//     normal_speed_task Inputs/csp_transfer_main_drives.SD41700_drv.channel_a.process_data_input.status_parametrization_level <-> AT 1/Status parametrization level
//     normal_speed_task Inputs/csp_transfer_main_drives.SD41700_drv.channel_a.process_data_input.warning_active <-> AT 1/Device control: Status word[2]
//     normal_speed_task Inputs/csp_transfer_main_drives.SD41700_drv.channel_b.process_data_input.status_parametrization_level <-> AT 1/Status parametrization level
//   SFI_CasePacker Instance <-> Transfer EtherCAT Master/Slot 57 (EK1100)/SPLC40210
//     highest_speed_task Inputs/csp_transfer_main_safety_drives_SD41100.chA_smes_sis.safely_closed_input.status <-> StandardInputs/SD41100.csp_transfer_main_safety_drives_SD41100chA_smes_sissafely_closed_inputstatus_31
//     highest_speed_task Inputs/csp_transfer_main_safety_drives_SD41300.chA_smes_sis.safely_closed_input.status <-> StandardInputs/SD41300.csp_transfer_main_safety_drives_SD41300chA_smes_sissafely_closed_inputstatus_61
//     highest_speed_task Inputs/csp_transfer_main_safety_drives_SD41400.chA_smes_sis.safely_closed_input.status <-> StandardInputs/SD41400.csp_transfer_main_safety_drives_SD41400chA_smes_sissafely_closed_inputstatus_69
//     highest_speed_task Inputs/csp_transfer_main_safety_drives_SD41500.chA_smes_sis.safely_closed_input.status <-> StandardInputs/SD41500.csp_transfer_main_safety_drives_SD41500chA_smes_sissafely_closed_inputstatus_77
//     highest_speed_task Inputs/csp_transfer_main_safety_drives_SD41100.chB_smes_sis.safely_closed_input.status <-> StandardInputs/SD41100.csp_transfer_main_safety_drives_SD41100chB_smes_sissafely_closed_inputstatus_32
//     highest_speed_task Inputs/csp_transfer_main_safety_drives_SD41300.chB_smes_sis.safely_closed_input.status <-> StandardInputs/SD41300.csp_transfer_main_safety_drives_SD41300chB_smes_sissafely_closed_inputstatus_62
//     highest_speed_task Inputs/csp_transfer_main_safety_drives_SD41400.chB_smes_sis.safely_closed_input.status <-> StandardInputs/SD41400.csp_transfer_main_safety_drives_SD41400chB_smes_sissafely_closed_inputstatus_70
//     highest_speed_task Inputs/csp_transfer_main_safety_drives_SD41500.chB_smes_sis.safely_closed_input.status <-> StandardInputs/SD41500.csp_transfer_main_safety_drives_SD41500chB_smes_sissafely_closed_inputstatus_78
//     highest_speed_task Inputs/csp_transfer_main_safety_guards.sis.safely_closed_input.status <-> StandardInputs/Guards.csp_transfer_main_safety_guardssissafely_closed_inputstatus_124
//     low_speed_task Inputs/csp_transfer_main_safety_accUChange.sig.group_info_data.info_data <-> TwinSAFE Group Info Data/AccUChange_STO Info Data
//     low_speed_task Inputs/csp_transfer_main_safety_accUChange.sis.discrepancy_input.status <-> StandardInputs/AccUChange_STO.csp_transfer_main_safety_accUChangesisdiscrepancy_inputstatus_169
//     low_speed_task Inputs/csp_transfer_main_safety_accUChange.sis.safely_closed_input.status <-> StandardInputs/AccUChange_STO.csp_transfer_main_safety_accUChangesissafely_closed_inputstatus_162
//     low_speed_task Inputs/csp_transfer_main_safety_drives_PS41020.sig.group_info_data.info_data <-> TwinSAFE Group Info Data/DrivesRackPowerSupply Info Data
//     low_speed_task Inputs/csp_transfer_main_safety_drives_PS41020.sig.safety_group_fb_err_input.status <-> StandardInputs/DrivesRackPowerSupply.csp_transfer_main_safety_drives_PS41020sigsafety_group_fb_err_inputstatus_172
//     low_speed_task Inputs/csp_transfer_main_safety_drives_SD41200.chA_smes_sis.safely_closed_input.status <-> StandardInputs/SD41200.csp_transfer_main_safety_drives_SD41200chA_smes_sissafely_closed_inputstatus_50
//     low_speed_task Inputs/csp_transfer_main_safety_drives_SD41600.chA_smes_sis.safely_closed_input.status <-> StandardInputs/SD41600.csp_transfer_main_safety_drives_SD41600chA_smes_sissafely_closed_inputstatus_85
//     low_speed_task Inputs/csp_transfer_main_safety_drives_SD41700.chA_smes_sis.safely_closed_input.status <-> StandardInputs/SD41700.csp_transfer_main_safety_drives_SD41700chA_smes_sissafely_closed_inputstatus_93
//     low_speed_task Inputs/csp_transfer_main_safety_drives_SD41200.chB_smes_sis.safely_closed_input.status <-> StandardInputs/SD41200.csp_transfer_main_safety_drives_SD41200chB_smes_sissafely_closed_inputstatus_52
//     low_speed_task Inputs/csp_transfer_main_safety_drives_SD41600.chB_smes_sis.safely_closed_input.status <-> StandardInputs/SD41600.csp_transfer_main_safety_drives_SD41600chB_smes_sissafely_closed_inputstatus_86
//     low_speed_task Inputs/csp_transfer_main_safety_drives_SD41700.chB_smes_sis.safely_closed_input.status <-> StandardInputs/SD41700.csp_transfer_main_safety_drives_SD41700chB_smes_sissafely_closed_inputstatus_94
//     low_speed_task Inputs/csp_transfer_main_safety_drives_commonConfiguration.rack_smes_sis.safely_closed_input.status <-> StandardInputs/DrivesCommonConfiguration.csp_transfer_main_safety_drives_commonConfigurationrack_smes_sissafely_closed_inputstatus_28
//     low_speed_task Inputs/csp_transfer_main_safety_drives_commonConfiguration.sig.group_info_data.info_data <-> TwinSAFE Group Info Data/DrivesCommonConfiguration Info Data
//     low_speed_task Inputs/csp_transfer_main_safety_emergency.HMI_button_sio.protection_safely_closed_input.status <-> StandardInputs/Interface.csp_transfer_main_safety_emergencyHMI_button_stop_sioprotection_safely_closed_inputstatus_6
//     low_speed_task Inputs/csp_transfer_main_safety_emergency.delayed_sis.safely_closed_input.status <-> StandardInputs/EmergencyCircuit.csp_transfer_main_safety_emergencydelayed_sissafely_closed_inputstatus_111
//     low_speed_task Inputs/csp_transfer_main_safety_emergency.sig.group_info_data.info_data <-> TwinSAFE Group Info Data/EmergencyCircuit Info Data
//     low_speed_task Inputs/csp_transfer_main_safety_guards.delayed_sis.safely_closed_input.status <-> StandardInputs/Guards.csp_transfer_main_safety_guardsdelayed_sissafely_closed_inputstatus_114
//     low_speed_task Inputs/csp_transfer_main_safety_guards.sig.group_info_data.info_data <-> TwinSAFE Group Info Data/Guards Info Data
//     low_speed_task Inputs/csp_transfer_main_safety_guards.sio_door_3.protection_discrepancy_input.status <-> StandardInputs/Guards.csp_transfer_main_safety_guardssio_door_3protection_discrepancy_inputstatus_115
//     low_speed_task Inputs/csp_transfer_main_safety_guards.sio_door_4.protection_discrepancy_input.status <-> StandardInputs/Guards.csp_transfer_main_safety_guardssio_door_4protection_discrepancy_inputstatus_126
//     low_speed_task Inputs/csp_transfer_main_safety_guards.sio_door_5.protection_discrepancy_input.status <-> StandardInputs/Guards.csp_transfer_main_safety_guardssio_door_5protection_discrepancy_inputstatus_128
//     low_speed_task Inputs/csp_transfer_main_safety_guards.sio_door_6.protection_discrepancy_input.status <-> StandardInputs/Guards.csp_transfer_main_safety_guardssio_door_6protection_discrepancy_inputstatus_132
//     low_speed_task Inputs/csp_transfer_main_safety_guards.sio_door_7.protection_discrepancy_input.status <-> StandardInputs/Guards.csp_transfer_main_safety_guardssio_door_7protection_discrepancy_inputstatus_148
//     low_speed_task Inputs/csp_transfer_main_safety_guards.sio_door_8.protection_discrepancy_input.status <-> StandardInputs/Guards.csp_transfer_main_safety_guardssio_door_8protection_discrepancy_inputstatus_151
//     low_speed_task Inputs/csp_transfer_main_safety_guards.sio_door_3.safely_closed_and_locked_input.status <-> StandardInputs/Guards.csp_transfer_main_safety_guardssio_door_3safely_closed_and_locked_inputstatus_118
//     low_speed_task Inputs/csp_transfer_main_safety_guards.sio_door_4.safely_closed_and_locked_input.status <-> StandardInputs/Guards.csp_transfer_main_safety_guardssio_door_4safely_closed_and_locked_inputstatus_125
//     low_speed_task Inputs/csp_transfer_main_safety_guards.sio_door_5.safely_closed_and_locked_input.status <-> StandardInputs/Guards.csp_transfer_main_safety_guardssio_door_5safely_closed_and_locked_inputstatus_129
//     low_speed_task Inputs/csp_transfer_main_safety_guards.sio_door_6.safely_closed_and_locked_input.status <-> StandardInputs/Guards.csp_transfer_main_safety_guardssio_door_6safely_closed_and_locked_inputstatus_133
//     low_speed_task Inputs/csp_transfer_main_safety_guards.sio_door_7.safely_closed_and_locked_input.status <-> StandardInputs/Guards.csp_transfer_main_safety_guardssio_door_7safely_closed_and_locked_inputstatus_149
//     low_speed_task Inputs/csp_transfer_main_safety_guards.sio_door_8.safely_closed_and_locked_input.status <-> StandardInputs/Guards.csp_transfer_main_safety_guardssio_door_8safely_closed_and_locked_inputstatus_150
//     low_speed_task Inputs/csp_transfer_main_safety_guards.sio_door_3.safely_locked_input.status <-> StandardInputs/Guards.csp_transfer_main_safety_guardssio_door_3safely_locked_inputstatus_116
//     low_speed_task Inputs/csp_transfer_main_safety_guards.sio_door_4.safely_locked_input.status <-> StandardInputs/Guards.csp_transfer_main_safety_guardssio_door_4safely_locked_inputstatus_141
//     low_speed_task Inputs/csp_transfer_main_safety_guards.sio_door_5.safely_locked_input.status <-> StandardInputs/Guards.csp_transfer_main_safety_guardssio_door_5safely_locked_inputstatus_130
//     low_speed_task Inputs/csp_transfer_main_safety_guards.sio_door_6.safely_locked_input.status <-> StandardInputs/Guards.csp_transfer_main_safety_guardssio_door_6safely_locked_inputstatus_142
//     low_speed_task Inputs/csp_transfer_main_safety_guards.sio_door_7.safely_locked_input.status <-> StandardInputs/Guards.csp_transfer_main_safety_guardssio_door_7safely_locked_inputstatus_152
//     low_speed_task Inputs/csp_transfer_main_safety_guards.sio_door_8.safely_locked_input.status <-> StandardInputs/Guards.csp_transfer_main_safety_guardssio_door_8safely_locked_inputstatus_153
//     low_speed_task Inputs/csp_transfer_main_safety_token.sig.group_info_data.info_data <-> TwinSAFE Group Info Data/SafetyToken Info Data
//     low_speed_task Inputs/csp_transfer_main_safety_token.sio.protection_discrepancy_input.status <-> StandardInputs/SafetyToken.csp_transfer_main_safety_tokensioprotection_discrepancy_inputstatus_140
//     low_speed_task Inputs/csp_transfer_main_safety_token.sio.protection_safely_closed_input.status <-> StandardInputs/Interface.csp_transfer_main_safety_tokensioprotection_safely_closed_inputstatus_171
//     low_speed_task Inputs/csp_transfer_main_safety_token.sis.safely_closed_input.status <-> StandardInputs/SafetyToken.csp_transfer_main_safety_tokensissafely_closed_inputstatus_137
//     low_speed_task Outputs/csp_transfer_main_safety_accUChange.sig.safety_group_err_ack_output.status <-> StandardOutputs/AccUChange_STO.ErrorAcknowledgement_159
//     low_speed_task Outputs/csp_transfer_main_safety_accUChange.sig.safety_group_run_output.status <-> StandardOutputs/AccUChange_STO.Run_160
//     low_speed_task Outputs/csp_transfer_main_safety_accUChange.sis.open_output.status <-> StandardOutputs/AccUChange_STO.csp_transfer_main_safety_accUChangesisopen_outputstatus_161
//     low_speed_task Outputs/csp_transfer_main_safety_drives_PS41020.sig.safety_group_err_ack_output.status <-> StandardOutputs/DrivesRackPowerSupply.csp_transfer_main_safety_drives_PS41020sigsafety_group_err_ack_outputstatus_13
//     low_speed_task Outputs/csp_transfer_main_safety_drives_PS41020.sig.safety_group_run_output.status <-> StandardOutputs/DrivesRackPowerSupply.csp_transfer_main_safety_drives_PS41020sigsafety_group_run_outputstatus_14
//     low_speed_task Outputs/csp_transfer_main_safety_drives_SD41100.chA_smes_sis.open_output.status <-> StandardOutputs/SD41100.csp_transfer_main_safety_drives_SD41100chA_smes_sisopen_outputstatus_22
//     low_speed_task Outputs/csp_transfer_main_safety_drives_SD41200.chA_smes_sis.open_output.status <-> StandardOutputs/SD41200.csp_transfer_main_safety_drives_SD41200chA_smes_sisopen_outputstatus_49
//     low_speed_task Outputs/csp_transfer_main_safety_drives_SD41300.chA_smes_sis.open_output.status <-> StandardOutputs/SD41300.csp_transfer_main_safety_drives_SD41300chA_smes_sisopen_outputstatus_57
//     low_speed_task Outputs/csp_transfer_main_safety_drives_SD41400.chA_smes_sis.open_output.status <-> StandardOutputs/SD41400.csp_transfer_main_safety_drives_SD41400chA_smes_sisopen_outputstatus_65
//     low_speed_task Outputs/csp_transfer_main_safety_drives_SD41500.chA_smes_sis.open_output.status <-> StandardOutputs/SD41500.csp_transfer_main_safety_drives_SD41500chA_smes_sisopen_outputstatus_73
//     low_speed_task Outputs/csp_transfer_main_safety_drives_SD41600.chA_smes_sis.open_output.status <-> StandardOutputs/SD41600.csp_transfer_main_safety_drives_SD41600chA_smes_sisopen_outputstatus_81
//     low_speed_task Outputs/csp_transfer_main_safety_drives_SD41700.chA_smes_sis.open_output.status <-> StandardOutputs/SD41700.csp_transfer_main_safety_drives_SD41700chA_smes_sisopen_outputstatus_89
//     low_speed_task Outputs/csp_transfer_main_safety_drives_SD41100.chB_smes_sis.open_output.status <-> StandardOutputs/SD41100.csp_transfer_main_safety_drives_SD41100chB_smes_sisopen_outputstatus_23
//     low_speed_task Outputs/csp_transfer_main_safety_drives_SD41200.chB_smes_sis.open_output.status <-> StandardOutputs/SD41200.csp_transfer_main_safety_drives_SD41200chB_smes_sisopen_outputstatus_51
//     low_speed_task Outputs/csp_transfer_main_safety_drives_SD41300.chB_smes_sis.open_output.status <-> StandardOutputs/SD41300.csp_transfer_main_safety_drives_SD41300chB_smes_sisopen_outputstatus_58
//     low_speed_task Outputs/csp_transfer_main_safety_drives_SD41400.chB_smes_sis.open_output.status <-> StandardOutputs/SD41400.csp_transfer_main_safety_drives_SD41400chB_smes_sisopen_outputstatus_66
//     low_speed_task Outputs/csp_transfer_main_safety_drives_SD41500.chB_smes_sis.open_output.status <-> StandardOutputs/SD41500.csp_transfer_main_safety_drives_SD41500chB_smes_sisopen_outputstatus_74
//     low_speed_task Outputs/csp_transfer_main_safety_drives_SD41600.chB_smes_sis.open_output.status <-> StandardOutputs/SD41600.csp_transfer_main_safety_drives_SD41600chB_smes_sisopen_outputstatus_82
//     low_speed_task Outputs/csp_transfer_main_safety_drives_SD41700.chB_smes_sis.open_output.status <-> StandardOutputs/SD41700.csp_transfer_main_safety_drives_SD41700chB_smes_sisopen_outputstatus_90
//     low_speed_task Outputs/csp_transfer_main_safety_drives_commonConfiguration.rack_smes_sis.open_output.status <-> StandardOutputs/DrivesCommonConfiguration.csp_transfer_main_safety_drives_commonConfigurationrack_smes_sisopen_outputstatus_27
//     low_speed_task Outputs/csp_transfer_main_safety_drives_commonConfiguration.sig.safety_group_err_ack_output.status <-> StandardOutputs/DrivesCommonConfiguration.ErrorAcknowledgement_25
//     low_speed_task Outputs/csp_transfer_main_safety_drives_commonConfiguration.sig.safety_group_run_output.status <-> StandardOutputs/DrivesCommonConfiguration.Run_26
//     low_speed_task Outputs/csp_transfer_main_safety_emergency.delayed_sis.open_output.status <-> StandardOutputs/EmergencyCircuit.csp_transfer_main_safety_emergencydelayed_sisopen_outputstatus_110
//     low_speed_task Outputs/csp_transfer_main_safety_emergency.sig.safety_group_err_ack_output.status <-> StandardOutputs/EmergencyCircuit.csp_transfer_main_safety_emergencysigsafety_group_err_ack_outputstatus_1
//     low_speed_task Outputs/csp_transfer_main_safety_emergency.sig.safety_group_run_output.status <-> StandardOutputs/EmergencyCircuit.csp_transfer_main_safety_emergencysigsafety_group_run_outputstatus_2
//     low_speed_task Outputs/csp_transfer_main_safety_guards.delayed_sis.open_output.status <-> StandardOutputs/Guards.csp_transfer_main_safety_guardsdelayed_sisopen_outputstatus_119
//     low_speed_task Outputs/csp_transfer_main_safety_guards.sig.safety_group_err_ack_output.status <-> StandardOutputs/Guards.ErrorAcknowledgement_112
//     low_speed_task Outputs/csp_transfer_main_safety_guards.sig.safety_group_run_output.status <-> StandardOutputs/Guards.Run_113
//     low_speed_task Outputs/csp_transfer_main_safety_guards.sio_door_3.unlock_output.status <-> StandardOutputs/Guards.csp_transfer_main_safety_guardssio_door_3unlock_outputstatus_127
//     low_speed_task Outputs/csp_transfer_main_safety_guards.sio_door_4.unlock_output.status <-> StandardOutputs/Guards.csp_transfer_main_safety_guardssio_door_4unlock_outputstatus_143
//     low_speed_task Outputs/csp_transfer_main_safety_guards.sio_door_5.unlock_output.status <-> StandardOutputs/Guards.csp_transfer_main_safety_guardssio_door_5unlock_outputstatus_131
//     low_speed_task Outputs/csp_transfer_main_safety_guards.sio_door_6.unlock_output.status <-> StandardOutputs/Guards.csp_transfer_main_safety_guardssio_door_6unlock_outputstatus_144
//     low_speed_task Outputs/csp_transfer_main_safety_guards.sio_door_7.unlock_output.status <-> StandardOutputs/Guards.csp_transfer_main_safety_guardssio_door_7unlock_outputstatus_154
//     low_speed_task Outputs/csp_transfer_main_safety_guards.sio_door_8.unlock_output.status <-> StandardOutputs/Guards.csp_transfer_main_safety_guardssio_door_8unlock_outputstatus_155
//     low_speed_task Outputs/csp_transfer_main_safety_token.sig.safety_group_err_ack_output.status <-> StandardOutputs/SafetyToken.ErrorAcknowledgement_134
//     low_speed_task Outputs/csp_transfer_main_safety_token.sig.safety_group_run_output.status <-> StandardOutputs/SafetyToken.Run_135
//     low_speed_task Outputs/csp_transfer_main_safety_token.sis.open_output.status <-> StandardOutputs/SafetyToken.csp_transfer_main_safety_tokensisopen_outputstatus_138
//     normal_speed_task Inputs/csp_transfer_main_safety_drives_PS41020.sis.discrepancy_input.status <-> StandardInputs/DrivesRackPowerSupply.csp_transfer_main_safety_drives_PS41020sisdiscrepancy_inputstatus_24
//     normal_speed_task Inputs/csp_transfer_main_safety_drives_PS41020.sis.safely_closed_input.status <-> StandardInputs/DrivesRackPowerSupply.csp_transfer_main_safety_drives_PS41020sissafely_closed_inputstatus_16
//     normal_speed_task Inputs/csp_transfer_main_safety_drives_SD{41100..41700 step 100}.sig.group_info_data.info_data <-> TwinSAFE Group Info Data/SD{41100..41700 step 100} Info Data  (7 links)
//     normal_speed_task Inputs/csp_transfer_main_safety_drives_SD41100.sig.safety_group_com_err_input.status <-> StandardInputs/SD41100.csp_transfer_main_safety_drives_SD41100sigsafety_group_com_err_inputstatus_36
//     normal_speed_task Inputs/csp_transfer_main_safety_drives_SD41200.sig.safety_group_com_err_input.status <-> StandardInputs/SD41200.csp_transfer_main_safety_drives_SD41200sigsafety_group_com_err_inputstatus_53
//     normal_speed_task Inputs/csp_transfer_main_safety_drives_SD41300.sig.safety_group_com_err_input.status <-> StandardInputs/SD41300.csp_transfer_main_safety_drives_SD41300sigsafety_group_com_err_inputstatus_63
//     normal_speed_task Inputs/csp_transfer_main_safety_drives_SD41400.sig.safety_group_com_err_input.status <-> StandardInputs/SD41400.csp_transfer_main_safety_drives_SD41400sigsafety_group_com_err_inputstatus_71
//     normal_speed_task Inputs/csp_transfer_main_safety_drives_SD41500.sig.safety_group_com_err_input.status <-> StandardInputs/SD41500.csp_transfer_main_safety_drives_SD41500sigsafety_group_com_err_inputstatus_79
//     normal_speed_task Inputs/csp_transfer_main_safety_drives_SD41600.sig.safety_group_com_err_input.status <-> StandardInputs/SD41600.csp_transfer_main_safety_drives_SD41600sigsafety_group_com_err_inputstatus_88
//     normal_speed_task Inputs/csp_transfer_main_safety_drives_SD41700.sig.safety_group_com_err_input.status <-> StandardInputs/SD41700.csp_transfer_main_safety_drives_SD41700sigsafety_group_com_err_inputstatus_95
//     normal_speed_task Inputs/csp_transfer_main_safety_drives_SD41100.sig.safety_group_fb_err_input.status <-> StandardInputs/SD41100.csp_transfer_main_safety_drives_SD41100sigsafety_group_fb_err_inputstatus_35
//     normal_speed_task Inputs/csp_transfer_main_safety_drives_SD41200.sig.safety_group_fb_err_input.status <-> StandardInputs/SD41200.csp_transfer_main_safety_drives_SD41200sigsafety_group_fb_err_inputstatus_54
//     normal_speed_task Inputs/csp_transfer_main_safety_drives_SD41300.sig.safety_group_fb_err_input.status <-> StandardInputs/SD41300.csp_transfer_main_safety_drives_SD41300sigsafety_group_fb_err_inputstatus_64
//     normal_speed_task Inputs/csp_transfer_main_safety_drives_SD41400.sig.safety_group_fb_err_input.status <-> StandardInputs/SD41400.csp_transfer_main_safety_drives_SD41400sigsafety_group_fb_err_inputstatus_72
//     normal_speed_task Inputs/csp_transfer_main_safety_drives_SD41500.sig.safety_group_fb_err_input.status <-> StandardInputs/SD41500.csp_transfer_main_safety_drives_SD41500sigsafety_group_fb_err_inputstatus_80
//     normal_speed_task Inputs/csp_transfer_main_safety_drives_SD41600.sig.safety_group_fb_err_input.status <-> StandardInputs/SD41600.csp_transfer_main_safety_drives_SD41600sigsafety_group_fb_err_inputstatus_87
//     normal_speed_task Inputs/csp_transfer_main_safety_drives_SD41700.sig.safety_group_fb_err_input.status <-> StandardInputs/SD41700.csp_transfer_main_safety_drives_SD41700sigsafety_group_fb_err_inputstatus_96
//     normal_speed_task Inputs/csp_transfer_main_safety_emergency.HMI_button_sio.protection_discrepancy_input.status <-> StandardInputs/EmergencyCircuit.csp_transfer_main_safety_emergencyHMI_button_sioprotection_discrepancy_inputstatus_12
//     normal_speed_task Inputs/csp_transfer_main_safety_emergency.sis.safely_closed_input.status <-> StandardInputs/EmergencyCircuit.csp_transfer_main_safety_emergencysissafely_closed_inputstatus_11
//     normal_speed_task Inputs/csp_transfer_main_safety_interface.SPLC40210_sig.group_info_data.info_data <-> TwinSAFE Group Info Data/Interface Info Data
//     normal_speed_task Inputs/csp_transfer_main_safety_interface._SD41100_drv_ChA.connection_info_data_interface.info_data <-> Connection Info Data/SD41100.SD41100_ChA_33 Info Data
//     normal_speed_task Inputs/csp_transfer_main_safety_interface._SD41200_drv_ChA.connection_info_data_interface.info_data <-> Connection Info Data/SD41200.SD41200_ChA_97 Info Data
//     normal_speed_task Inputs/csp_transfer_main_safety_interface._SD41300_drv_ChA.connection_info_data_interface.info_data <-> Connection Info Data/SD41300.SD41300_ChA_99 Info Data
//     normal_speed_task Inputs/csp_transfer_main_safety_interface._SD41400_drv_ChA.connection_info_data_interface.info_data <-> Connection Info Data/SD41400.SD41400_ChA_101 Info Data
//     normal_speed_task Inputs/csp_transfer_main_safety_interface._SD41500_drv_ChA.connection_info_data_interface.info_data <-> Connection Info Data/SD41500.SD41500_ChA_103 Info Data
//     normal_speed_task Inputs/csp_transfer_main_safety_interface._SD41600_drv_ChA.connection_info_data_interface.info_data <-> Connection Info Data/SD41600.SD41600_ChA_105 Info Data
//     normal_speed_task Inputs/csp_transfer_main_safety_interface._SD41700_drv_ChA.connection_info_data_interface.info_data <-> Connection Info Data/SD41700.SD41700_ChA_107 Info Data
//     normal_speed_task Inputs/csp_transfer_main_safety_interface._SD41100_drv_ChB.connection_info_data_interface.info_data <-> Connection Info Data/SD41100.SD41100_ChB_34 Info Data
//     normal_speed_task Inputs/csp_transfer_main_safety_interface._SD41200_drv_ChB.connection_info_data_interface.info_data <-> Connection Info Data/SD41200.SD41200_ChB_98 Info Data
//     normal_speed_task Inputs/csp_transfer_main_safety_interface._SD41300_drv_ChB.connection_info_data_interface.info_data <-> Connection Info Data/SD41300.SD41300_ChB_100 Info Data
//     normal_speed_task Inputs/csp_transfer_main_safety_interface._SD41400_drv_ChB.connection_info_data_interface.info_data <-> Connection Info Data/SD41400.SD41400_ChB_102 Info Data
//     normal_speed_task Inputs/csp_transfer_main_safety_interface._SD41500_drv_ChB.connection_info_data_interface.info_data <-> Connection Info Data/SD41500.SD41500_ChB_104 Info Data
//     normal_speed_task Inputs/csp_transfer_main_safety_interface._SD41600_drv_ChB.connection_info_data_interface.info_data <-> Connection Info Data/SD41600.SD41600_ChB_106 Info Data
//     normal_speed_task Inputs/csp_transfer_main_safety_interface._SD41700_drv_ChB.connection_info_data_interface.info_data <-> Connection Info Data/SD41700.SD41700_ChB_108 Info Data
//     normal_speed_task Inputs/csp_transfer_main_safety_interface._SPLC40210Slot59.connection_info_data_interface.info_data <-> Connection Info Data/Interface.SPLC40210Slot59_156 Info Data
//     normal_speed_task Inputs/csp_transfer_main_safety_interface._SPLC40210Slot60.connection_info_data_interface.info_data <-> Connection Info Data/Interface.SPLC40210Slot60_109 Info Data
//     normal_speed_task Inputs/csp_transfer_main_safety_interface._SPLC40210Slot61.connection_info_data_interface.info_data <-> Connection Info Data/Interface.SPLC40210Slot61_136 Info Data
//     normal_speed_task Inputs/csp_transfer_main_safety_interface._SPLC40210Slot68.connection_info_data_interface.info_data <-> Connection Info Data/Interface.SPLC40210Slot68_145 Info Data
//     normal_speed_task Inputs/csp_transfer_main_safety_interface._SPLC40210Slot70.connection_info_data_interface.info_data <-> Connection Info Data/Interface.SPLC40210Slot70_146 Info Data
//     normal_speed_task Inputs/csp_transfer_main_safety_interface._SPLC40210Slot72.connection_info_data_interface.info_data <-> Connection Info Data/Interface.SPLC40210Slot72_147 Info Data
//     normal_speed_task Outputs/csp_transfer_main_safety_drives_PS41020.sis.open_output.status <-> StandardOutputs/DrivesRackPowerSupply.csp_transfer_main_safety_drives_PS41020sisopen_outputstatus_15
//     normal_speed_task Outputs/csp_transfer_main_safety_drives_SD41100.sig.safety_group_err_ack_output.status <-> StandardOutputs/SD41100.ErrorAcknowledgement_18
//     normal_speed_task Outputs/csp_transfer_main_safety_drives_SD41200.sig.safety_group_err_ack_output.status <-> StandardOutputs/SD41200.ErrorAcknowledgement_37
//     normal_speed_task Outputs/csp_transfer_main_safety_drives_SD41300.sig.safety_group_err_ack_output.status <-> StandardOutputs/SD41300.ErrorAcknowledgement_39
//     normal_speed_task Outputs/csp_transfer_main_safety_drives_SD41400.sig.safety_group_err_ack_output.status <-> StandardOutputs/SD41400.ErrorAcknowledgement_41
//     normal_speed_task Outputs/csp_transfer_main_safety_drives_SD41500.sig.safety_group_err_ack_output.status <-> StandardOutputs/SD41500.ErrorAcknowledgement_43
//     normal_speed_task Outputs/csp_transfer_main_safety_drives_SD41600.sig.safety_group_err_ack_output.status <-> StandardOutputs/SD41600.ErrorAcknowledgement_45
//     normal_speed_task Outputs/csp_transfer_main_safety_drives_SD41700.sig.safety_group_err_ack_output.status <-> StandardOutputs/SD41700.ErrorAcknowledgement_47
//     normal_speed_task Outputs/csp_transfer_main_safety_drives_SD41100.sig.safety_group_run_output.status <-> StandardOutputs/SD41100.Run_19
//     normal_speed_task Outputs/csp_transfer_main_safety_drives_SD41200.sig.safety_group_run_output.status <-> StandardOutputs/SD41200.Run_38
//     normal_speed_task Outputs/csp_transfer_main_safety_drives_SD41300.sig.safety_group_run_output.status <-> StandardOutputs/SD41300.Run_40
//     normal_speed_task Outputs/csp_transfer_main_safety_drives_SD41400.sig.safety_group_run_output.status <-> StandardOutputs/SD41400.Run_42
//     normal_speed_task Outputs/csp_transfer_main_safety_drives_SD41500.sig.safety_group_run_output.status <-> StandardOutputs/SD41500.Run_44
//     normal_speed_task Outputs/csp_transfer_main_safety_drives_SD41600.sig.safety_group_run_output.status <-> StandardOutputs/SD41600.Run_46
//     normal_speed_task Outputs/csp_transfer_main_safety_drives_SD41700.sig.safety_group_run_output.status <-> StandardOutputs/SD41700.Run_48
//     normal_speed_task Outputs/csp_transfer_main_safety_emergency.sis.open_output.status <-> StandardOutputs/EmergencyCircuit.csp_transfer_main_safety_emergencysisopen_outputstatus_7
//     normal_speed_task Outputs/csp_transfer_main_safety_guards.sis.open_output.status <-> StandardOutputs/Guards.csp_transfer_main_safety_guardssisopen_outputstatus_120
//     normal_speed_task Outputs/csp_transfer_main_safety_interface.SPLC40210_sig.safety_group_err_ack_output.status <-> StandardOutputs/Interface.csp_transfer_main_safety_interfaceSPLC40210_sigsafety_group_err_ack_outputstatus_3
//     normal_speed_task Outputs/csp_transfer_main_safety_interface.SPLC40210_sig.safety_group_run_output.status <-> StandardOutputs/Interface.csp_transfer_main_safety_interfaceSPLC40210_sigsafety_group_run_outputstatus_4
//   SFI_CasePacker Instance <-> Transfer EtherCAT Master/Slot 57 (EK1100)/Slot 75 (EL1819)
//     low_speed_task Inputs/csp_transfer_main.temperature_fault_di.field.status <-> Channel 5/Input
//     low_speed_task Inputs/csp_transfer_main_safety_guards.sio_door_3.protection_safely_closed_input.status <-> Channel 1/Input
//     low_speed_task Inputs/csp_transfer_main_safety_guards.sio_door_4.protection_safely_closed_input.status <-> Channel 2/Input
//     low_speed_task Inputs/csp_transfer_main_safety_guards.sio_door_5.protection_safely_closed_input.status <-> Channel 3/Input
//     low_speed_task Inputs/csp_transfer_main_safety_guards.sio_door_6.protection_safely_closed_input.status <-> Channel 4/Input
//     low_speed_task Inputs/csp_transfer_main_safety_guards.sio_door_7.protection_safely_closed_input.status <-> Channel 6/Input
//     low_speed_task Inputs/csp_transfer_main_safety_guards.sio_door_8.protection_safely_closed_input.status <-> Channel 7/Input
//   SFI_CasePacker Instance <-> Transfer EtherCAT Master/Slot 57 (EK1100)/Slot 77 (EL2008)
//     normal_speed_task Outputs/csp_transfer_main_services.lights_on_do.field.status <-> Channel 2/Output
//     normal_speed_task Outputs/csp_transfer_main_services_pushbuttons.emergency_close_lamp_do.field.status <-> Channel 1/Output
//   SFI_CasePacker Instance <-> NC-Task 1 SAF/Axes/csp_case_closing_ls_horizontal_axis
//     highest_speed_task Inputs/csp_case_closing_ls_horizontal.axis.ax_ref.NcToPlc <-> Outputs/ToPlc
//     highest_speed_task Outputs/csp_case_closing_ls_horizontal.axis.ax_ref.PlcToNc <-> Inputs/FromPlc
//   SFI_CasePacker Instance <-> NC-Task 1 SAF/Axes/csp_case_closing_ls_lower_axis
//     highest_speed_task Inputs/csp_case_closing_ls_lower.axis.ax_ref.NcToPlc <-> Outputs/ToPlc
//     highest_speed_task Outputs/csp_case_closing_ls_lower.axis.ax_ref.PlcToNc <-> Inputs/FromPlc
//   SFI_CasePacker Instance <-> NC-Task 1 SAF/Axes/csp_case_closing_ls_upper_axis
//     highest_speed_task Inputs/csp_case_closing_ls_upper.axis.ax_ref.NcToPlc <-> Outputs/ToPlc
//     highest_speed_task Outputs/csp_case_closing_ls_upper.axis.ax_ref.PlcToNc <-> Inputs/FromPlc
//   SFI_CasePacker Instance <-> NC-Task 1 SAF/Axes/csp_case_closing_os_horizontal_axis
//     highest_speed_task Inputs/csp_case_closing_os_horizontal.axis.ax_ref.NcToPlc <-> Outputs/ToPlc
//     highest_speed_task Outputs/csp_case_closing_os_horizontal.axis.ax_ref.PlcToNc <-> Inputs/FromPlc
//   SFI_CasePacker Instance <-> NC-Task 1 SAF/Axes/csp_case_closing_os_lower_axis
//     highest_speed_task Inputs/csp_case_closing_os_lower.axis.ax_ref.NcToPlc <-> Outputs/ToPlc
//     highest_speed_task Outputs/csp_case_closing_os_lower.axis.ax_ref.PlcToNc <-> Inputs/FromPlc
//   SFI_CasePacker Instance <-> NC-Task 1 SAF/Axes/csp_case_closing_os_upper_axis
//     highest_speed_task Inputs/csp_case_closing_os_upper.axis.ax_ref.NcToPlc <-> Outputs/ToPlc
//     highest_speed_task Outputs/csp_case_closing_os_upper.axis.ax_ref.PlcToNc <-> Inputs/FromPlc
//   SFI_CasePacker Instance <-> NC-Task 1 SAF/Axes/csp_case_discharge_accU_depth_axis
//     normal_speed_task Inputs/csp_case_feed_reject_accU_depth.axis.ax_ref.NcToPlc <-> Outputs/ToPlc
//     normal_speed_task Outputs/csp_case_feed_reject_accU_depth.axis.ax_ref.PlcToNc <-> Inputs/FromPlc
//   SFI_CasePacker Instance <-> NC-Task 1 SAF/Axes/csp_case_discharge_reject_belt_axis
//     normal_speed_task Inputs/csp_case_discharge_reject_belt.axis.ax_ref.NcToPlc <-> Outputs/ToPlc
//     normal_speed_task Outputs/csp_case_discharge_reject_belt.axis.ax_ref.PlcToNc <-> Inputs/FromPlc
//   SFI_CasePacker Instance <-> NC-Task 1 SAF/Axes/csp_case_discharge_speedBelt_ls_axis
//     highest_speed_task Inputs/csp_case_discharge_speedBelt_ls.axis.ax_ref.NcToPlc <-> Outputs/ToPlc
//     highest_speed_task Outputs/csp_case_discharge_speedBelt_ls.axis.ax_ref.PlcToNc <-> Inputs/FromPlc
//   SFI_CasePacker Instance <-> NC-Task 1 SAF/Axes/csp_case_discharge_speedBelt_os_axis
//     highest_speed_task Inputs/csp_case_discharge_speedBelt_os.axis.ax_ref.NcToPlc <-> Outputs/ToPlc
//     highest_speed_task Outputs/csp_case_discharge_speedBelt_os.axis.ax_ref.PlcToNc <-> Inputs/FromPlc
//   SFI_CasePacker Instance <-> NC-Task 1 SAF/Axes/csp_case_fc_ls_lower_follower_axis
//     highest_speed_task Inputs/csp_case_fc_ls_lower_follower.axis.ax_ref.NcToPlc <-> Outputs/ToPlc
//     highest_speed_task Outputs/csp_case_fc_ls_lower_follower.axis.ax_ref.PlcToNc <-> Inputs/FromPlc
//   SFI_CasePacker Instance <-> NC-Task 1 SAF/Axes/csp_case_fc_ls_lower_spreader_axis
//     highest_speed_task Inputs/csp_case_fc_ls_lower_spreader.axis.ax_ref.NcToPlc <-> Outputs/ToPlc
//     highest_speed_task Outputs/csp_case_fc_ls_lower_spreader.axis.ax_ref.PlcToNc <-> Inputs/FromPlc
//   SFI_CasePacker Instance <-> NC-Task 1 SAF/Axes/csp_case_fc_ls_lower_trailingCloser_axis
//     highest_speed_task Inputs/csp_case_fc_ls_lower_trailingCloser.axis.ax_ref.NcToPlc <-> Outputs/ToPlc
//     highest_speed_task Outputs/csp_case_fc_ls_lower_trailingCloser.axis.ax_ref.PlcToNc <-> Inputs/FromPlc
//   SFI_CasePacker Instance <-> NC-Task 1 SAF/Axes/csp_case_fc_ls_upper_follower_axis
//     highest_speed_task Inputs/csp_case_fc_ls_upper_follower.axis.ax_ref.NcToPlc <-> Outputs/ToPlc
//     highest_speed_task Outputs/csp_case_fc_ls_upper_follower.axis.ax_ref.PlcToNc <-> Inputs/FromPlc
//   SFI_CasePacker Instance <-> NC-Task 1 SAF/Axes/csp_case_fc_ls_upper_leadingMinorCloser_axis
//     highest_speed_task Inputs/csp_case_fc_ls_upper_leadingMinorCloser.axis.ax_ref.NcToPlc <-> Outputs/ToPlc
//     highest_speed_task Outputs/csp_case_fc_ls_upper_leadingMinorCloser.axis.ax_ref.PlcToNc <-> Inputs/FromPlc
//   SFI_CasePacker Instance <-> NC-Task 1 SAF/Axes/csp_case_fc_ls_upper_leadingMinorCloser_virtual_axis
//     highest_speed_task Inputs/csp_case_fc_ls_upper_leadingMinorCloser_virtual.axis.ax_ref.NcToPlc <-> Outputs/ToPlc
//     highest_speed_task Outputs/csp_case_fc_ls_upper_leadingMinorCloser_virtual.axis.ax_ref.PlcToNc <-> Inputs/FromPlc
//   SFI_CasePacker Instance <-> NC-Task 1 SAF/Axes/csp_case_fc_ls_upper_spreader_axis
//     highest_speed_task Inputs/csp_case_fc_ls_upper_spreader.axis.ax_ref.NcToPlc <-> Outputs/ToPlc
//     highest_speed_task Outputs/csp_case_fc_ls_upper_spreader.axis.ax_ref.PlcToNc <-> Inputs/FromPlc
//   SFI_CasePacker Instance <-> NC-Task 1 SAF/Axes/csp_case_fc_os_lower_follower_axis
//     highest_speed_task Inputs/csp_case_fc_os_lower_follower.axis.ax_ref.NcToPlc <-> Outputs/ToPlc
//     highest_speed_task Outputs/csp_case_fc_os_lower_follower.axis.ax_ref.PlcToNc <-> Inputs/FromPlc
//   SFI_CasePacker Instance <-> NC-Task 1 SAF/Axes/csp_case_fc_os_lower_spreader_axis
//     highest_speed_task Inputs/csp_case_fc_os_lower_spreader.axis.ax_ref.NcToPlc <-> Outputs/ToPlc
//     highest_speed_task Outputs/csp_case_fc_os_lower_spreader.axis.ax_ref.PlcToNc <-> Inputs/FromPlc
//   SFI_CasePacker Instance <-> NC-Task 1 SAF/Axes/csp_case_fc_os_upper_follower_axis
//     highest_speed_task Inputs/csp_case_fc_os_upper_follower.axis.ax_ref.NcToPlc <-> Outputs/ToPlc
//     highest_speed_task Outputs/csp_case_fc_os_upper_follower.axis.ax_ref.PlcToNc <-> Inputs/FromPlc
//   SFI_CasePacker Instance <-> NC-Task 1 SAF/Axes/csp_case_fc_os_upper_spreader_axis
//     highest_speed_task Inputs/csp_case_fc_os_upper_spreader.axis.ax_ref.NcToPlc <-> Outputs/ToPlc
//     highest_speed_task Outputs/csp_case_fc_os_upper_spreader.axis.ax_ref.PlcToNc <-> Inputs/FromPlc
//   SFI_CasePacker Instance <-> NC-Task 1 SAF/Axes/csp_case_feed_arm_Tilt
//     highest_speed_task Inputs/csp_case_feed_kinematic_tilt.axis.ax_ref.NcToPlc <-> Outputs/ToPlc
//     highest_speed_task Outputs/csp_case_feed_kinematic_tilt.axis.ax_ref.PlcToNc <-> Inputs/FromPlc
//   SFI_CasePacker Instance <-> NC-Task 1 SAF/Axes/csp_case_feed_arm_X
//     highest_speed_task Inputs/csp_case_feed_kinematic_x.axis.ax_ref.NcToPlc <-> Outputs/ToPlc
//     highest_speed_task Outputs/csp_case_feed_kinematic_x.axis.ax_ref.PlcToNc <-> Inputs/FromPlc
//   SFI_CasePacker Instance <-> NC-Task 1 SAF/Axes/csp_case_feed_arm_Y
//     highest_speed_task Inputs/csp_case_feed_kinematic_y.axis.ax_ref.NcToPlc <-> Outputs/ToPlc
//     highest_speed_task Outputs/csp_case_feed_kinematic_y.axis.ax_ref.PlcToNc <-> Inputs/FromPlc
//   SFI_CasePacker Instance <-> NC-Task 1 SAF/Axes/csp_case_feed_arm_elbow_axis
//     highest_speed_task Inputs/csp_case_feed_arm_elbow.axis.ax_ref.NcToPlc <-> Outputs/ToPlc
//     highest_speed_task Outputs/csp_case_feed_arm_elbow.axis.ax_ref.PlcToNc <-> Inputs/FromPlc
//   SFI_CasePacker Instance <-> NC-Task 1 SAF/Axes/csp_case_feed_arm_shoulder_axis
//     highest_speed_task Inputs/csp_case_feed_arm_shoulder.axis.ax_ref.NcToPlc <-> Outputs/ToPlc
//     highest_speed_task Outputs/csp_case_feed_arm_shoulder.axis.ax_ref.PlcToNc <-> Inputs/FromPlc
//   SFI_CasePacker Instance <-> NC-Task 1 SAF/Axes/csp_case_feed_arm_wrist_axis
//     highest_speed_task Inputs/csp_case_feed_arm_wrist.axis.ax_ref.NcToPlc <-> Outputs/ToPlc
//     highest_speed_task Outputs/csp_case_feed_arm_wrist.axis.ax_ref.PlcToNc <-> Inputs/FromPlc
//   SFI_CasePacker Instance <-> NC-Task 1 SAF/Axes/csp_case_feed_magazine_accU_lsDepth_axis
//     normal_speed_task Inputs/csp_case_feed_magazine_accU_lsDepth.axis.ax_ref.NcToPlc <-> Outputs/ToPlc
//     normal_speed_task Outputs/csp_case_feed_magazine_accU_lsDepth.axis.ax_ref.PlcToNc <-> Inputs/FromPlc
//   SFI_CasePacker Instance <-> NC-Task 1 SAF/Axes/csp_case_feed_magazine_accU_osDepth_axis
//     normal_speed_task Inputs/csp_case_feed_magazine_accU_osDepth.axis.ax_ref.NcToPlc <-> Outputs/ToPlc
//     normal_speed_task Outputs/csp_case_feed_magazine_accU_osDepth.axis.ax_ref.PlcToNc <-> Inputs/FromPlc
//   SFI_CasePacker Instance <-> NC-Task 1 SAF/Axes/csp_case_feed_magazine_ls_belt_axis
//     normal_speed_task Inputs/csp_case_feed_magazine_ls_belt.axis.ax_ref.NcToPlc <-> Outputs/ToPlc
//     normal_speed_task Outputs/csp_case_feed_magazine_ls_belt.axis.ax_ref.PlcToNc <-> Inputs/FromPlc
//   SFI_CasePacker Instance <-> NC-Task 1 SAF/Axes/csp_case_feed_magazine_os_belt_axis
//     normal_speed_task Inputs/csp_case_feed_magazine_os_belt.axis.ax_ref.NcToPlc <-> Outputs/ToPlc
//     normal_speed_task Outputs/csp_case_feed_magazine_os_belt.axis.ax_ref.PlcToNc <-> Inputs/FromPlc
//   SFI_CasePacker Instance <-> NC-Task 1 SAF/Axes/csp_case_feed_reject_belt_lower_axis
//     low_speed_task Inputs/csp_case_feed_reject_belt_lower.axis.ax_ref.NcToPlc <-> Outputs/ToPlc
//     low_speed_task Outputs/csp_case_feed_reject_belt_lower.axis.ax_ref.PlcToNc <-> Inputs/FromPlc
//   SFI_CasePacker Instance <-> NC-Task 1 SAF/Axes/csp_case_feed_reject_belt_upper_axis
//     low_speed_task Inputs/csp_case_feed_reject_belt_upper.axis.ax_ref.NcToPlc <-> Outputs/ToPlc
//     low_speed_task Outputs/csp_case_feed_reject_belt_upper.axis.ax_ref.PlcToNc <-> Inputs/FromPlc
//   SFI_CasePacker Instance <-> NC-Task 1 SAF/Axes/csp_case_feed_shuttle_accU_depth_axis
//     normal_speed_task Inputs/csp_case_feed_shuttle_accU_depth.axis.ax_ref.NcToPlc <-> Outputs/ToPlc
//     normal_speed_task Outputs/csp_case_feed_shuttle_accU_depth.axis.ax_ref.PlcToNc <-> Inputs/FromPlc
//   SFI_CasePacker Instance <-> NC-Task 1 SAF/Axes/csp_case_feed_shuttle_horizontal_axis
//     highest_speed_task Inputs/csp_case_feed_shuttle_horizontal.axis.ax_ref.NcToPlc <-> Outputs/ToPlc
//     highest_speed_task Outputs/csp_case_feed_shuttle_horizontal.axis.ax_ref.PlcToNc <-> Inputs/FromPlc
//   SFI_CasePacker Instance <-> NC-Task 1 SAF/Axes/csp_case_feed_shuttle_vertical_axis
//     highest_speed_task Inputs/csp_case_feed_shuttle_vertical.axis.ax_ref.NcToPlc <-> Outputs/ToPlc
//     highest_speed_task Outputs/csp_case_feed_shuttle_vertical.axis.ax_ref.PlcToNc <-> Inputs/FromPlc
//   SFI_CasePacker Instance <-> NC-Task 1 SAF/Axes/csp_case_feed_virtualMaster_axis
//     highest_speed_task Inputs/csp_case_feed_virtualMaster.axis.ax_ref.NcToPlc <-> Outputs/ToPlc
//     highest_speed_task Outputs/csp_case_feed_virtualMaster.axis.ax_ref.PlcToNc <-> Inputs/FromPlc
//   SFI_CasePacker Instance <-> NC-Task 1 SAF/Axes/csp_case_glue_ls_accU_lowerPosition_axis
//     normal_speed_task Inputs/csp_case_glue_ls_accU_lowerPosition.axis.ax_ref.NcToPlc <-> Outputs/ToPlc
//     normal_speed_task Outputs/csp_case_glue_ls_accU_lowerPosition.axis.ax_ref.PlcToNc <-> Inputs/FromPlc
//   SFI_CasePacker Instance <-> NC-Task 1 SAF/Axes/csp_case_glue_ls_accU_upperPosition_axis
//     normal_speed_task Inputs/csp_case_glue_ls_accU_upperPosition.axis.ax_ref.NcToPlc <-> Outputs/ToPlc
//     normal_speed_task Outputs/csp_case_glue_ls_accU_upperPosition.axis.ax_ref.PlcToNc <-> Inputs/FromPlc
//   SFI_CasePacker Instance <-> NC-Task 1 SAF/Axes/csp_case_glue_os_accU_Width_axis
//     normal_speed_task Inputs/csp_case_glue_os_accU_width.axis.ax_ref.NcToPlc <-> Outputs/ToPlc
//     normal_speed_task Outputs/csp_case_glue_os_accU_width.axis.ax_ref.PlcToNc <-> Inputs/FromPlc
//   SFI_CasePacker Instance <-> NC-Task 1 SAF/Axes/csp_case_glue_os_accU_lowerPosition_axis
//     normal_speed_task Inputs/csp_case_glue_os_accU_lowerPosition.axis.ax_ref.NcToPlc <-> Outputs/ToPlc
//     normal_speed_task Outputs/csp_case_glue_os_accU_lowerPosition.axis.ax_ref.PlcToNc <-> Inputs/FromPlc
//   SFI_CasePacker Instance <-> NC-Task 1 SAF/Axes/csp_case_glue_os_accU_upperPosition_axis
//     normal_speed_task Inputs/csp_case_glue_os_accU_upperPosition.axis.ax_ref.NcToPlc <-> Outputs/ToPlc
//     normal_speed_task Outputs/csp_case_glue_os_accU_upperPosition.axis.ax_ref.PlcToNc <-> Inputs/FromPlc
//   SFI_CasePacker Instance <-> NC-Task 1 SAF/Axes/csp_case_loader_guide_accU_width_axis
//     normal_speed_task Inputs/csp_case_loader_guide_accU_width.axis.ax_ref.NcToPlc <-> Outputs/ToPlc
//     normal_speed_task Outputs/csp_case_loader_guide_accU_width.axis.ax_ref.PlcToNc <-> Inputs/FromPlc
//   SFI_CasePacker Instance <-> NC-Task 1 SAF/Axes/csp_case_loader_guide_downstream_axis
//     highest_speed_task Inputs/csp_case_loader_guide_downstream.axis.ax_ref.NcToPlc <-> Outputs/ToPlc
//     highest_speed_task Outputs/csp_case_loader_guide_downstream.axis.ax_ref.PlcToNc <-> Inputs/FromPlc
//   SFI_CasePacker Instance <-> NC-Task 1 SAF/Axes/csp_case_loader_guide_length_axis
//     low_speed_task Inputs/csp_case_loader_guide_length.axis.ax_ref.NcToPlc <-> Outputs/ToPlc
//     low_speed_task Outputs/csp_case_loader_guide_length.axis.ax_ref.PlcToNc <-> Inputs/FromPlc
//   SFI_CasePacker Instance <-> NC-Task 1 SAF/Axes/csp_case_loader_guide_upstream_axis
//     highest_speed_task Inputs/csp_case_loader_guide_upstream.axis.ax_ref.NcToPlc <-> Outputs/ToPlc
//     highest_speed_task Outputs/csp_case_loader_guide_upstream.axis.ax_ref.PlcToNc <-> Inputs/FromPlc
//   SFI_CasePacker Instance <-> NC-Task 1 SAF/Axes/csp_case_loader_pusher_axis
//     highest_speed_task Inputs/csp_case_loader_pusher.axis.ax_ref.NcToPlc <-> Outputs/ToPlc
//     highest_speed_task Outputs/csp_case_loader_pusher.axis.ax_ref.PlcToNc <-> Inputs/FromPlc
//   SFI_CasePacker Instance <-> NC-Task 1 SAF/Axes/csp_case_loader_virtualMaster
//     highest_speed_task Inputs/csp_case_loader_virtualMaster.axis.ax_ref.NcToPlc <-> Outputs/ToPlc
//     highest_speed_task Outputs/csp_case_loader_virtualMaster.axis.ax_ref.PlcToNc <-> Inputs/FromPlc
//   SFI_CasePacker Instance <-> NC-Task 1 SAF/Axes/csp_case_tr_accU_depth_axis
//     normal_speed_task Inputs/csp_case_tr_accU_depth.axis.ax_ref.NcToPlc <-> Outputs/ToPlc
//     normal_speed_task Outputs/csp_case_tr_accU_depth.axis.ax_ref.PlcToNc <-> Inputs/FromPlc
//   SFI_CasePacker Instance <-> NC-Task 1 SAF/Axes/csp_case_tr_accU_ls_width_axis
//     normal_speed_task Inputs/csp_case_tr_accU_ls_width.axis.ax_ref.NcToPlc <-> Outputs/ToPlc
//     normal_speed_task Outputs/csp_case_tr_accU_ls_width.axis.ax_ref.PlcToNc <-> Inputs/FromPlc
//   SFI_CasePacker Instance <-> NC-Task 1 SAF/Axes/csp_case_tr_accU_os_width_axis
//     normal_speed_task Inputs/csp_case_tr_accU_os_width.axis.ax_ref.NcToPlc <-> Outputs/ToPlc
//     normal_speed_task Outputs/csp_case_tr_accU_os_width.axis.ax_ref.PlcToNc <-> Inputs/FromPlc
//   SFI_CasePacker Instance <-> NC-Task 1 SAF/Axes/csp_case_tr_accU_virtualMaster
//     low_speed_task Inputs/csp_case_tr_accU_virtualMaster.axis.ax_ref.NcToPlc <-> Outputs/ToPlc
//     low_speed_task Outputs/csp_case_tr_accU_virtualMaster.axis.ax_ref.PlcToNc <-> Inputs/FromPlc
//   SFI_CasePacker Instance <-> NC-Task 1 SAF/Axes/csp_case_tr_squaring_ls_leading_axis
//     highest_speed_task Inputs/csp_case_tr_squaring_ls_leading.axis.ax_ref.NcToPlc <-> Outputs/ToPlc
//     highest_speed_task Outputs/csp_case_tr_squaring_ls_leading.axis.ax_ref.PlcToNc <-> Inputs/FromPlc
//   SFI_CasePacker Instance <-> NC-Task 1 SAF/Axes/csp_case_tr_squaring_ls_trailing_axis
//     highest_speed_task Inputs/csp_case_tr_squaring_ls_trailing.axis.ax_ref.NcToPlc <-> Outputs/ToPlc
//     highest_speed_task Outputs/csp_case_tr_squaring_ls_trailing.axis.ax_ref.PlcToNc <-> Inputs/FromPlc
//   SFI_CasePacker Instance <-> NC-Task 1 SAF/Axes/csp_case_tr_squaring_os_leading_axis
//     highest_speed_task Inputs/csp_case_tr_squaring_os_leading.axis.ax_ref.NcToPlc <-> Outputs/ToPlc
//     highest_speed_task Outputs/csp_case_tr_squaring_os_leading.axis.ax_ref.PlcToNc <-> Inputs/FromPlc
//   SFI_CasePacker Instance <-> NC-Task 1 SAF/Axes/csp_case_tr_squaring_os_trailing_axis
//     highest_speed_task Inputs/csp_case_tr_squaring_os_trailing.axis.ax_ref.NcToPlc <-> Outputs/ToPlc
//     highest_speed_task Outputs/csp_case_tr_squaring_os_trailing.axis.ax_ref.PlcToNc <-> Inputs/FromPlc
//   SFI_CasePacker Instance <-> NC-Task 1 SAF/Axes/csp_case_transport_accU_depth_axis
//     normal_speed_task Inputs/csp_case_transport_accU_depth.axis.ax_ref.NcToPlc <-> Outputs/ToPlc
//     normal_speed_task Outputs/csp_case_transport_accU_depth.axis.ax_ref.PlcToNc <-> Inputs/FromPlc
//   SFI_CasePacker Instance <-> NC-Task 1 SAF/Axes/csp_case_transport_accU_virtualMaster
//     low_speed_task Inputs/csp_case_transport_accU_virtualMaster.axis.ax_ref.NcToPlc <-> Outputs/ToPlc
//     low_speed_task Outputs/csp_case_transport_accU_virtualMaster.axis.ax_ref.PlcToNc <-> Inputs/FromPlc
//   SFI_CasePacker Instance <-> NC-Task 1 SAF/Axes/csp_case_transport_ls_leading_axis
//     highest_speed_task Inputs/csp_case_transport_ls_leading.axis.ax_ref.NcToPlc <-> Outputs/ToPlc
//     highest_speed_task Outputs/csp_case_transport_ls_leading.axis.ax_ref.PlcToNc <-> Inputs/FromPlc
//   SFI_CasePacker Instance <-> NC-Task 1 SAF/Axes/csp_case_transport_ls_trailing_axis
//     highest_speed_task Inputs/csp_case_transport_ls_trailing.axis.ax_ref.NcToPlc <-> Outputs/ToPlc
//     highest_speed_task Outputs/csp_case_transport_ls_trailing.axis.ax_ref.PlcToNc <-> Inputs/FromPlc
//   SFI_CasePacker Instance <-> NC-Task 1 SAF/Axes/csp_case_transport_os_leading_axis
//     highest_speed_task Inputs/csp_case_transport_os_leading.axis.ax_ref.NcToPlc <-> Outputs/ToPlc
//     highest_speed_task Outputs/csp_case_transport_os_leading.axis.ax_ref.PlcToNc <-> Inputs/FromPlc
//   SFI_CasePacker Instance <-> NC-Task 1 SAF/Axes/csp_case_transport_os_trailing_axis
//     highest_speed_task Inputs/csp_case_transport_os_trailing.axis.ax_ref.NcToPlc <-> Outputs/ToPlc
//     highest_speed_task Outputs/csp_case_transport_os_trailing.axis.ax_ref.PlcToNc <-> Inputs/FromPlc
//   SFI_CasePacker Instance <-> NC-Task 1 SAF/Axes/csp_case_transport_virtualMaster_axis
//     highest_speed_task Inputs/csp_case_transport_virtualMaster.axis.ax_ref.NcToPlc <-> Outputs/ToPlc
//     highest_speed_task Outputs/csp_case_transport_virtualMaster.axis.ax_ref.PlcToNc <-> Inputs/FromPlc
//   SFI_CasePacker Instance <-> NC-Task 1 SAF/Axes/csp_case_virtualMaster_axis
//     highest_speed_task Inputs/csp_case_virtualMaster.axis.ax_ref.NcToPlc <-> Outputs/ToPlc
//     highest_speed_task Outputs/csp_case_virtualMaster.axis.ax_ref.PlcToNc <-> Inputs/FromPlc
//   SFI_CasePacker Instance <-> NC-Task 1 SAF/Axes/csp_main_motorization_virtualManager_axis
//     highest_speed_task Inputs/csp_main_motorization_virtualManager.axis.ax_ref.NcToPlc <-> Outputs/ToPlc
//     highest_speed_task Outputs/csp_main_motorization_virtualManager.axis.ax_ref.PlcToNc <-> Inputs/FromPlc
//   SFI_CasePacker Instance <-> NC-Task 1 SAF/Axes/csp_main_motorization_virtualManager_machine_periodicity_axis
//     highest_speed_task Inputs/csp_main_motorization_virtualManager.machine_periodicity_axis.ax_ref.NcToPlc <-> Outputs/ToPlc
//     highest_speed_task Outputs/csp_main_motorization_virtualManager.machine_periodicity_axis.ax_ref.PlcToNc <-> Inputs/FromPlc
//   SFI_CasePacker Instance <-> NC-Task 1 SAF/Axes/csp_main_motorization_virtualManager_virtual_master_test
//     highest_speed_task Inputs/csp_main_motorization_virtualManager.virtual_master_test.ax_ref.NcToPlc <-> Outputs/ToPlc
//     highest_speed_task Outputs/csp_main_motorization_virtualManager.virtual_master_test.ax_ref.PlcToNc <-> Inputs/FromPlc
//   SFI_CasePacker Instance <-> NC-Task 1 SAF/Axes/csp_transfer_accumulator_accU_convDepth_axis
//     normal_speed_task Inputs/csp_transfer_accumulator_accU_convDepth.axis.ax_ref.NcToPlc <-> Outputs/ToPlc
//     normal_speed_task Outputs/csp_transfer_accumulator_accU_convDepth.axis.ax_ref.PlcToNc <-> Inputs/FromPlc
//   SFI_CasePacker Instance <-> NC-Task 1 SAF/Axes/csp_transfer_accumulator_accU_depth_axis
//     normal_speed_task Inputs/csp_transfer_accumulator_accU_depth.axis.ax_ref.NcToPlc <-> Outputs/ToPlc
//     normal_speed_task Outputs/csp_transfer_accumulator_accU_depth.axis.ax_ref.PlcToNc <-> Inputs/FromPlc
//   SFI_CasePacker Instance <-> NC-Task 1 SAF/Axes/csp_transfer_accumulator_accU_topRailLength_axis
//     low_speed_task Inputs/csp_transfer_accumulator_accU_topRailLength.axis.ax_ref.NcToPlc <-> Outputs/ToPlc
//     low_speed_task Outputs/csp_transfer_accumulator_accU_topRailLength.axis.ax_ref.PlcToNc <-> Inputs/FromPlc
//   SFI_CasePacker Instance <-> NC-Task 1 SAF/Axes/csp_transfer_accumulator_accU_topRailWidth_axis
//     low_speed_task Inputs/csp_transfer_accumulator_accU_topRailWidth.axis.ax_ref.NcToPlc <-> Outputs/ToPlc
//     low_speed_task Inputs/csp_transfer_accumulator_accU_topRailWidth.axis.hard_increments.value <-> Enc/Outputs/Out/nDataOut1
//     low_speed_task Outputs/csp_transfer_accumulator_accU_topRailWidth.axis.ax_ref.PlcToNc <-> Inputs/FromPlc
//   SFI_CasePacker Instance <-> NC-Task 1 SAF/Axes/csp_transfer_accumulator_accU_virtualMaster
//     low_speed_task Inputs/csp_transfer_accumulator_accU_virtualMaster.axis.ax_ref.NcToPlc <-> Outputs/ToPlc
//     low_speed_task Outputs/csp_transfer_accumulator_accU_virtualMaster.axis.ax_ref.PlcToNc <-> Inputs/FromPlc
//   SFI_CasePacker Instance <-> NC-Task 1 SAF/Axes/csp_transfer_accumulator_belt_axis
//     highest_speed_task Inputs/csp_transfer_accumulator_belt.axis.ax_ref.NcToPlc <-> Outputs/ToPlc
//     highest_speed_task Outputs/csp_transfer_accumulator_belt.axis.ax_ref.PlcToNc <-> Inputs/FromPlc
//   SFI_CasePacker Instance <-> NC-Task 1 SAF/Axes/csp_transfer_accumulator_finger_ls_axis
//     highest_speed_task Inputs/csp_transfer_accumulator_finger_ls.axis.ax_ref.NcToPlc <-> Outputs/ToPlc
//     highest_speed_task Outputs/csp_transfer_accumulator_finger_ls.axis.ax_ref.PlcToNc <-> Inputs/FromPlc
//   SFI_CasePacker Instance <-> NC-Task 1 SAF/Axes/csp_transfer_accumulator_finger_os_axis
//     highest_speed_task Inputs/csp_transfer_accumulator_finger_os.axis.ax_ref.NcToPlc <-> Outputs/ToPlc
//     highest_speed_task Outputs/csp_transfer_accumulator_finger_os.axis.ax_ref.PlcToNc <-> Inputs/FromPlc
//   SFI_CasePacker Instance <-> NC-Task 1 SAF/Axes/csp_transfer_accumulator_lift_axis
//     highest_speed_task Inputs/csp_transfer_accumulator_lift.axis.ax_ref.NcToPlc <-> Outputs/ToPlc
//     highest_speed_task Outputs/csp_transfer_accumulator_lift.axis.ax_ref.PlcToNc <-> Inputs/FromPlc
//   SFI_CasePacker Instance <-> NC-Task 1 SAF/Axes/csp_transfer_accumulator_virtualMaster_axis
//     highest_speed_task Inputs/csp_transfer_accumulator_virtualMaster.axis.ax_ref.NcToPlc <-> Outputs/ToPlc
//     highest_speed_task Outputs/csp_transfer_accumulator_virtualMaster.axis.ax_ref.PlcToNc <-> Inputs/FromPlc
//   SFI_CasePacker Instance <-> NC-Task 1 SAF/Axes/csp_transfer_crosspusher_follower_axis
//     highest_speed_task Inputs/csp_transfer_crosspusher_follower.axis.ax_ref.NcToPlc <-> Outputs/ToPlc
//     highest_speed_task Outputs/csp_transfer_crosspusher_follower.axis.ax_ref.PlcToNc <-> Inputs/FromPlc
//   SFI_CasePacker Instance <-> NC-Task 1 SAF/Axes/csp_transfer_crosspusher_horizontal_axis
//     highest_speed_task Inputs/csp_transfer_crosspusher_horizontal.axis.ax_ref.NcToPlc <-> Outputs/ToPlc
//     highest_speed_task Outputs/csp_transfer_crosspusher_horizontal.axis.ax_ref.PlcToNc <-> Inputs/FromPlc
//   SFI_CasePacker Instance <-> NC-Task 1 SAF/Axes/csp_transfer_crosspusher_vertical_axis
//     highest_speed_task Inputs/csp_transfer_crosspusher_vertical.axis.ax_ref.NcToPlc <-> Outputs/ToPlc
//     highest_speed_task Outputs/csp_transfer_crosspusher_vertical.axis.ax_ref.PlcToNc <-> Inputs/FromPlc
//   SFI_CasePacker Instance <-> NC-Task 1 SAF/Axes/csp_transfer_crosspusher_virtualMaster_axis
//     highest_speed_task Inputs/csp_transfer_crosspusher_virtualMaster.axis.ax_ref.NcToPlc <-> Outputs/ToPlc
//     highest_speed_task Outputs/csp_transfer_crosspusher_virtualMaster.axis.ax_ref.PlcToNc <-> Inputs/FromPlc
//   SFI_CasePacker Instance <-> NC-Task 1 SAF/Axes/csp_transfer_infeed_accU_depth_axis
//     normal_speed_task Inputs/csp_transfer_infeed_accU_depth.axis.ax_ref.NcToPlc <-> Outputs/ToPlc
//     normal_speed_task Outputs/csp_transfer_infeed_accU_depth.axis.ax_ref.PlcToNc <-> Inputs/FromPlc
//   SFI_CasePacker Instance <-> NC-Task 1 SAF/Axes/csp_transfer_infeed_accU_waterfallAdjust_axis
//     normal_speed_task Inputs/csp_transfer_infeed_accU_waterfallAdjust.axis.ax_ref.NcToPlc <-> Outputs/ToPlc
//     normal_speed_task Outputs/csp_transfer_infeed_accU_waterfallAdjust.axis.ax_ref.PlcToNc <-> Inputs/FromPlc
//   SFI_CasePacker Instance <-> NC-Task 1 SAF/Axes/csp_transfer_infeed_accumulation_belt_axis
//     highest_speed_task Inputs/csp_transfer_infeed_accumulation_belt.axis.ax_ref.NcToPlc <-> Outputs/ToPlc
//     highest_speed_task Outputs/csp_transfer_infeed_accumulation_belt.axis.ax_ref.PlcToNc <-> Inputs/FromPlc
//   SFI_CasePacker Instance <-> NC-Task 1 SAF/Axes/csp_transfer_infeed_metering_belt_axis
//     highest_speed_task Inputs/csp_transfer_infeed_metering_belt.axis.ax_ref.NcToPlc <-> Outputs/ToPlc
//     highest_speed_task Outputs/csp_transfer_infeed_metering_belt.axis.ax_ref.PlcToNc <-> Inputs/FromPlc
//   SFI_CasePacker Instance <-> NC-Task 1 SAF/Axes/csp_transfer_infeed_reject_pusher_axis
//     highest_speed_task Inputs/csp_transfer_infeed_reject_pusher.axis.ax_ref.NcToPlc <-> Outputs/ToPlc
//     highest_speed_task Outputs/csp_transfer_infeed_reject_pusher.axis.ax_ref.PlcToNc <-> Inputs/FromPlc
//   SFI_CasePacker Instance <-> NC-Task 1 SAF/Axes/csp_transfer_infeed_reject_virtualMaster
//     highest_speed_task Inputs/csp_transfer_infeed_reject_virtualMaster.axis.ax_ref.NcToPlc <-> Outputs/ToPlc
//     highest_speed_task Outputs/csp_transfer_infeed_reject_virtualMaster.axis.ax_ref.PlcToNc <-> Inputs/FromPlc
//   SFI_CasePacker Instance <-> NC-Task 1 SAF/Axes/csp_transfer_infeed_waterfall_belt_axis
//     highest_speed_task Inputs/csp_transfer_infeed_waterfall_belt.axis.ax_ref.NcToPlc <-> Outputs/ToPlc
//     highest_speed_task Outputs/csp_transfer_infeed_waterfall_belt.axis.ax_ref.PlcToNc <-> Inputs/FromPlc
//   SFI_CasePacker Instance <-> NC-Task 1 SAF/Axes/csp_transfer_upstacker_downstream_axis
//     highest_speed_task Inputs/csp_transfer_upstacker_downstream.axis.ax_ref.NcToPlc <-> Outputs/ToPlc
//     highest_speed_task Outputs/csp_transfer_upstacker_downstream.axis.ax_ref.PlcToNc <-> Inputs/FromPlc
//   SFI_CasePacker Instance <-> NC-Task 1 SAF/Axes/csp_transfer_upstacker_upstream_axis
//     highest_speed_task Inputs/csp_transfer_upstacker_upstream.axis.ax_ref.NcToPlc <-> Outputs/ToPlc
//     highest_speed_task Outputs/csp_transfer_upstacker_upstream.axis.ax_ref.PlcToNc <-> Inputs/FromPlc
//   SFI_CasePacker Instance <-> NC-Task 1 SAF/Axes/csp_transfer_upstacker_virtualMaster_axis
//     highest_speed_task Inputs/csp_transfer_upstacker_virtualMaster.axis.ax_ref.NcToPlc <-> Outputs/ToPlc
//     highest_speed_task Outputs/csp_transfer_upstacker_virtualMaster.axis.ax_ref.PlcToNc <-> Inputs/FromPlc
//   SFI_CasePacker Instance <-> NC-Task 1 SAF/Axes/csp_transfer_virtualMaster_axis
//     highest_speed_task Inputs/csp_transfer_virtualMaster.axis.ax_ref.NcToPlc <-> Outputs/ToPlc
//     highest_speed_task Outputs/csp_transfer_virtualMaster.axis.ax_ref.PlcToNc <-> Inputs/FromPlc
//   SFI_CasePacker Instance <-> NC-Task 1 SAF/Kinematics
//     highest_speed_task Inputs/csp_case_feed_kinematic.in_stKinToPlc <-> Outputs/ToPlc

CONFIGURATION SFI_CasePacker
    RESOURCE PLC ON TwinCAT3
        TASK highest_speed_task(INTERVAL := T#2ms, PRIORITY := 6);
        TASK lowest_speed_task(INTERVAL := T#48ms, PRIORITY := 16);
        TASK low_speed_task(INTERVAL := T#16ms, PRIORITY := 14);
        TASK normal_speed_task(INTERVAL := T#8ms, PRIORITY := 12);
        PROGRAM _highest WITH highest_speed_task : _highest;
        PROGRAM _lowest WITH lowest_speed_task : _lowest;
        PROGRAM _low WITH low_speed_task : _low;
        PROGRAM _normal WITH normal_speed_task : _normal;
    END_RESOURCE
END_CONFIGURATION

// ---- Application/auxiliary_counters_code_enum.TcDUT
TYPE auxiliary_counters_code_enum :
(
	INFEED_REJECT_BARCODE				:= 1,
	INFEED_REJECT_HIGH_LOAD				:= 2,
	CROSSPUSHER_REJECT_LOW_LOAD			:= 3,
	CROSSPUSHER_REJECT_HIGH_LOAD		:= 4,
	CASE_FEED_REJECT					:= 5,
	TOTAL_UNITS							:= 7	
);
END_TYPE

// ---- Application/CSP/cam_table_enum.TcTLEO
TYPE cam_table_enum :(
    NO_SELECTED_CAM 											:= 0,
	
	(* GENERIC - PERIODIC*)
	
	LINEAR_CAM													:= 1,
	FORWARD_CAM													:= 4, (*csp_transfer_infeed_reject_pusher_axis, csp_transfer_upstacker_virtualMaster*)
	BACKWARD_CAM												:= 5, (*csp_case_discharge_speedBelt_os, csp_case_discharge_speedBelt_ls*)
	DWELL_CAM													:= 6, (*csp_case_loader_guide_length, csp_transfer_upstacker_virtualMaster*)
	GEAR_CAM													:= 18,

	(*	CASE PACKER CAMS *)
	CASE_TRANSPORT_RUN_CAM										:= 13, (*csp_case_transport_os_leading,csp_case_transport_os_trailing, csp_case_transport_ls_leading, csp_case_transport_ls_trailing*)
	CASE_CLOSING_UPPER_RUN_CAM									:= 8,  (*csp_case_closing_os_upper, csp_case_closing_ls_upper,*)
	CASE_CLOSING_LOWER_RUN_CAM									:= 14, (*csp_case_closing_os_lower, csp_case_closing_ls_lower*) 
	CASE_CLOSING_HORIZONTAL_RUN_CAM								:= 15, (*csp_case_closing_os_horizontal, csp_case_ls_closing_horizontal*)
	CASE_FC_LEADINGCLOSER_LS_RUN_CAM							:= 16, (*csp_case_fc_ls_upper_leadingMinorCloser*)
	CASE_FC_TRAILINGCLOSER_LS_RUN_CAM							:= 22, (*csp_case_fc_ls_lower_trailingCloser*)
	CASE_LOADER_PUSHER_RUN_CAM									:= 20, (*csp_case_loader_pusher*)
	CASE_LOADER_GUIDE_RUN_CAM									:= 21, (*csp_case_loader_guide_upstream, csp_case_loader_guide_downstream*)
	CASE_FC_SPREADER_RUN_CAM									:= 23, (*csp_case_fc_os_upper_spreader, csp_case_fc_ls_upper_spreader, csp_case_fc_ls_lower_spreader*)
	CASE_FC_FOLLOWER_RUN_CAM									:= 24, (*csp_case_fc_os_upper_follower, csp_case_fc_ls_upper_follower, csp_case_fc_ls_lower_follower*)  
	CASE_TR_SQUARING_TRAILING_RUN_CAM							:= 25, (*csp_case_tr_squaring_os_trailing, csp_case_tr_squaring_ls_trailing*)
	CASE_TR_SQUARING_LEADING_RUN_CAM							:= 26, (*csp_case_tr_squaring_os_leading, csp_case_tr_squaring_ls_leading*)
	CASE_FC_TRAILINGCLOSER_OS_RUN_CAM							:= 31, (*csp_case_fc_os_lower_trailingCloser*)
	CASE_FEED_SHUTTLE_HORIZONTAL_RUN_CAM						:= 32, (*csp_case_feed_shuttle_virtual_master*)
	CASE_FEED_SHUTTLE_VERTICAL_RUN_CAM							:= 33, (*csp_case_feed_shuttle_virtual_master*)
	CASE_DISCHARGE_SPEED_BELTS_RUN_CAM							:= 37, (*csp_case_discharge_speed_belts*)
	CASE_FEED_KINEMATIC_X_RUN_CAM								:= 2, (*csp_case_feed_shuttle_virtual_master*)
	CASE_FEED_KINEMATIC_Y_RUN_CAM								:= 3, (*csp_case_feed_shuttle_virtual_master*)
	CASE_FEED_KINEMATIC_TILT_RUN_CAM							:= 7, (*csp_case_feed_shuttle_virtual_master*)
	
	CASE_FC_OS_LOWER_SPREADER_RUN_CAM							:= 901, (* csp_case_fc_os_lower_spreader *)
	CASE_FC_OS_LOWER_FOLLOWER_RUN_CAM							:= 902, (* csp_case_fc_os_lower_follower *)
	
		(* --------------------- TRANSFER CAMS --------------------- *)
	(*INFEED*)
	TRANSFER_INFEED_REJECT_RUN_CAM								:= 60,

	(*UPSTACKER*)
	TRANSFER_UPSTACKER_DOWNSTREAM_RUN_CAM						:= 81, (*OLD 30  csp_transfer_upstacker_downstream*)
	TRANSFER_UPSTACKER_DOWNSTREAM_PHASING_STEP1_CAM				:= 84, (*OLD 40  csp_transfer_upstacker_downstream CAM_ID TO BE CHANGED->+20*)
	TRANSFER_UPSTACKER_DOWNSTREAM_PHASING_STEP2_CAM				:= 85, (*OLD 41  csp_transfer_upstacker_downstream CAM_ID TO BE CHANGEDv*)
	TRANSFER_UPSTACKER_UPSTREAM_RUN_CAM							:= 80, (*OLD 44  csp_transfer_upstacker_upstream CAM_ID TO BE CHANGED->+20*)
	TRANSFER_UPSTACKER_UPSTREAM_PHASING_STEP1_CAM				:= 82, (*OLD 42  csp_transfer_upstacker_upstream CAM_ID TO BE CHANGED->+20*)
	TRANSFER_UPSTACKER_UPSTREAM_PHASING_STEP2_CAM				:= 83, (*OLD 43  csp_transfer_upstacker_upstream CAM_ID TO BE CHANGED->+20*)
	TRANSFER_UPSTACKER_VIRTUAL_STOP_CAM							:= 61, (*OLD 51   csp_transfer_upstacker_virtualMaster CAM_ID TO BE CHANGED->+20*)
	TRANSFER_UPSTACKER_VIRTUAL_START_CAM						:= 62, (*OLD 52   csp_transfer_upstacker_virtualMaster CAM_ID TO BE CHANGED->+20*)

	(*CROSSPUSHER*)
	TRANSFER_CROSSPUSHER_HORIZONTAL_TO_UPSTACKER				:= 100,
	TRANSFER_CROSSPUSHER_HORIZONTAL_TO_LOAD						:= 101,
	TRANSFER_CROSSPUSHER_FOLLOWER_TO_UPSTACK_TO_LOAD			:= 202, //102,
	TRANSFER_CROSSPUSHER_VERTICAL_RUN							:= 103,
	
	(*ACCUMULATOR*)
	TRANSFER_UPSTACKER_FINGER_RUN_CAM							:= 34, (*csp_transfer_accumulator_finger_os CAM_ID TO BE CHANGED->+20*)
	TRANSFER_ACCUMULATOR_LIFT_RUN								:= 104,
	TRANSFER_ACCUMULATOR_BELT_RUN								:= 105,
	
	(* LEADING MINOR CLOSER *)
	CASE_FC_LEADING_MINOR_RUN_DOWNSTREAM_RUN_CAM				:= 10,
	CASE_FC_LEADING_MINOR_RUN_UPSTREAM_RUN_CAM					:= 9

    ) := NO_SELECTED_CAM;
END_TYPE

// ---- Application/CSP/Case/Closing/csp_case_closing_constant_struct.TcDUT
TYPE csp_case_closing_constant_struct :
STRUCT
	(*BELT Info*)
	MIN_VELOCITY_MMpSEC:						LREAL := 100;
	MAX_VELOCITY_MMpSEC:						LREAL := 1000;
	MAX_ACCELERATION_MMpSEC2:					LREAL := 10000;
	MAX_DECELERATION_MMpSEC2:					LREAL := 10000;
	MAX_JERK_MMpSEC3:							LREAL := 1000000;
	RUNNING_ACCELERATION_MMMpSEC2:				LREAL := 3000;
	RUNNING_DECELERATION_MMpSEC2:				LREAL := 3000;
	MAX_FOLLOWING_ERROR_MM:						LREAL := 100;
	
	RUNNING_JERK_MMpSEC3:						LREAL := 1000000;
	MOTOR_MAX_VELOCITY_DEGPS:					LREAL := 9600;
	MOTOR_MAX_ACCELERATION_DEGPS2:				LREAL := 4800;
	MOTOR_MAX_DECELERATION_DEGPS2:				LREAL := 4800;
	MOTOR_MAX_JERK_DEGPS3:						LREAL := 100000000; 
	MOTOR_MAX_FOLLOWING_ERROR_DEG:				LREAL := 2;
END_STRUCT
END_TYPE

// ---- Application/CSP/Case/Closing/csp_case_closing_status_enum.TcDUT
TYPE csp_case_closing_status_enum :
(
	CSP_CASE_CLOSING_STATUS_NOT_INITIALIZED 							:=  0,
	CSP_CASE_CLOSING_STATUS_DISABLED 									:=  10,
	CSP_CASE_CLOSING_STATUS_ENABLE_REQUEST 								:=  20,
	CSP_CASE_CLOSING_STATUS_ENABLING 									:=  30,
	CSP_CASE_CLOSING_STATUS_ENABLED 									:=  40,
	CSP_CASE_CLOSING_STATUS_CHANGE_OVER_MODE							:=  45,
	CSP_CASE_CLOSING_STATUS_CHANGE_OVER_MODE_MOVE_DONE					:= 445,
	CSP_CASE_CLOSING_STATUS_CHANGE_OVER_RFID_MOVE_TO_CHECK				:=  46,
	CSP_CASE_CLOSING_STATUS_CHANGE_OVER_RFID_CHECK_SENSOR				:=  47,
	CSP_CASE_CLOSING_STATUS_CHANGE_OVER_RFID_MOVE_BACK					:=  48,
	CSP_CASE_CLOSING_STATUS_CHANGE_OVER_RFID_COMPLETE					:=  49,
	CSP_CASE_CLOSING_STATUS_HOME_REQUEST								:=  50,
	CSP_CASE_CLOSING_STATUS_HOMING										:=  60,
	CSP_CASE_CLOSING_STATUS_HOME_DONE									:=  70,
	CSP_CASE_CLOSING_STATUS_CALCULATING_SLAVE_POSITION					:=  90,
	CSP_CASE_CLOSING_STATUS_WAITING_SLAVE_ENGAGE						:= 100,
	CSP_CASE_CLOSING_STATUS_PHASE_REQUEST								:= 140,
	CSP_CASE_CLOSING_STATUS_PHASING										:= 150,
	CSP_CASE_CLOSING_STATUS_PHASED										:= 160,
	CSP_CASE_CLOSING_STATUS_CAM_ENGAGED_REQ								:= 170,
	CSP_CASE_CLOSING_STATUS_AXIS_ENGAGE_VERIFY							:= 180,
	CSP_CASE_CLOSING_STATUS_CAM_ENGAGED									:= 190,
	CSP_CASE_CLOSING_STATUS_CAM_TABLE_READ								:= 195,
	CSP_CASE_CLOSING_STATUS_CALCULATE_SLAVE_POSITION_REQUEST			:= 196,
	CSP_CASE_CLOSING_STATUS_READY										:= 197,
	CSP_CASE_CLOSING_STATUS_RUNNING										:= 200,
	CSP_CASE_CLOSING_STATUS_MOVING										:= 205,
	CSP_CASE_CLOSING_STATUS_DISENGAGE_REQUEST							:= 210,
	CSP_CASE_CLOSING_STATUS_DISENGAGING									:= 211,	
	CSP_CASE_CLOSING_STATUS_STOP_REQUEST 								:= 500,
	CSP_CASE_CLOSING_STATUS_DISABLE_REQUEST 							:= 530,
	CSP_CASE_CLOSING_STATUS_DISABLING 									:= 540
) := CSP_CASE_CLOSING_STATUS_NOT_INITIALIZED;
END_TYPE

// ---- Application/CSP/Case/Closing/csp_case_closing_rfid_status_enum.TcDUT
TYPE csp_case_closing_rfid_status_enum :
(
	CSP_CASE_CLOSING_RFID_STATUS_START									:= 5,
	CSP_CASE_CLOSING_RFID_STATUS_ENABLED								:= 6,
	CSP_CASE_CLOSING_RFID_STATUS_PADDLES_START							:= 10,
	CSP_CASE_CLOSING_RFID_STATUS_VERIFY_AXIS_SAFE_POS					:= 15,
	CSP_CASE_CLOSING_RFID_STATUS_UPPER_START 							:= 20,
	CSP_CASE_CLOSING_RFID_STATUS_UPPER_VERIFY_AXIS_POS					:= 25,
	CSP_CASE_CLOSING_RFID_STATUS_UPPER_READ_START						:= 30,
	CSP_CASE_CLOSING_RFID_STATUS_UPPER_READ_CHECK_RESULT				:= 35,
	CSP_CASE_CLOSING_RFID_STATUS_UPPER_RETURN_TO_SAFE_POS				:= 40,
	CSP_CASE_CLOSING_RFID_STATUS_UPPER_READ_DONE						:= 45,
	
	CSP_CASE_CLOSING_RFID_STATUS_LOWER_START 							:= 50,
	CSP_CASE_CLOSING_RFID_STATUS_LOWER_VERIFY_AXIS_POS					:= 55,
	CSP_CASE_CLOSING_RFID_STATUS_LOWER_READ_START						:= 60,
	CSP_CASE_CLOSING_RFID_STATUS_LOWER_READ_CHECK_RESULT				:= 65,
	CSP_CASE_CLOSING_RFID_STATUS_LOWER_RETURN_TO_SAFE_POS				:= 70,
	CSP_CASE_CLOSING_RFID_STATUS_LOWER_READ_DONE						:= 75,
	
	
	CSP_CASE_CLOSING_RFID_STATUS_VERIFY_VALUES							:= 100,
		
	CSP_CASE_CLOSING_RFID_STATUS_COMPLETE								:= 220,
	
	CSP_CASE_CLOSING_RFID_STATUS_ERROR									:= 666,
			
	CSP_CASE_CLOSING_RFID_STATUS_WAITING								:= 900
	
) := CSP_CASE_CLOSING_RFID_STATUS_START;
END_TYPE

// ---- Application/CSP/Case/csp_case_connection_status_enum.TcDUT
TYPE csp_case_connection_status_enum :
(		
	CSP_CASE_STATUS_CONNECTION_START							:= 0,
	CSP_CASE_STATUS_CONNECTION_ENGAGE							:= 10,
	CSP_CASE_STATUS_CONNECTION_ENGAGED							:= 20,
	CSP_CASE_STATUS_CONNECTION_CHECK_CHANGE_CAM					:= 30,
	CSP_CASE_STATUS_CONNECTION_CHANGE_CAM						:= 40,
	CSP_CASE_STATUS_CONNECTION_WAIT_NEW_CAM						:= 50,
	CSP_CASE_STATUS_CONNECTION_DONE 							:= 900,
	CSP_CASE_STATUS_CONNECTION_ERROR 							:= 999
) := CSP_CASE_STATUS_CONNECTION_START;
END_TYPE

// ---- Application/CSP/Case/csp_case_phase_status_enum.TcDUT
TYPE csp_case_phase_status_enum :
(		
	CSP_CASE_PHASE_STATUS_START									:= 0,
	CSP_CASE_PHASE_STATUS_DISABLE 								:= 10,
	CSP_CASE_PHASE_STATUS_ENABLE 								:= 20,	
	CSP_CASE_PHASE_STATUS_ENABLED 								:= 30,
	CSP_CASE_PHASE_STATUS_CALCULATE_SLAVE_POSITION_REQUEST		:= 31,
	CSP_CASE_PHASE_STATUS_CALCULATING_SLAVE_POSITION			:= 32,
	CSP_CASE_PHASE_STATUS_REQUEST								:= 33,
	CSP_CASE_PHASE_STATUS_PHASING								:= 34,
	CSP_CASE_PHASE_STATUS_PHASED								:= 35,
	CSP_CASE_PHASE_STATUS_REDEFINE								:= 40,
	CSP_CASE_PHASE_STATUS_REDEFINED								:= 50,
	CSP_CASE_PHASE_STATUS_DONE 									:= 900,
	CSP_CASE_PHASE_STATUS_ERROR 								:= 999
) := CSP_CASE_PHASE_STATUS_START;
END_TYPE

// ---- Application/CSP/Case/csp_case_status_enum.TcDUT
TYPE csp_case_status_enum :
(
	CSP_CASE_STATUS_NOT_INITIALIZED 							:=  0,
	CSP_CASE_STATUS_DISABLED 									:=  10,
	CSP_CASE_STATUS_ENABLE_REQUEST 								:=  20,
	CSP_CASE_STATUS_ENABLING 									:=  30,
	CSP_CASE_STATUS_ENABLED 									:=  40,
	CSP_CASE_STATUS_HOME_REQUEST								:=  50,
	CSP_CASE_STATUS_HOMING										:=  60,
	CSP_CASE_STATUS_HOME_DONE									:=  70,
	CSP_CASE_STATUS_CALCULATING_SLAVE_POSITION					:=  90,
	CSP_CASE_STATUS_WAITING_SLAVE_ENGAGE						:= 100,
	CSP_CASE_STATUS_PHASE_REQUEST								:= 140,
	CSP_CASE_STATUS_PHASING										:= 150,
	CSP_CASE_STATUS_PHASED										:= 160,
	CSP_CASE_STATUS_CAM_ENGAGED_REQ								:= 170,
	CSP_CASE_STATUS_AXIS_ENGAGE_VERIFY							:= 180,
	CSP_CASE_STATUS_CAM_ENGAGED									:= 190,
	CSP_CASE_STATUS_CAM_TABLE_READ								:= 195,
	CSP_CASE_STATUS_CALCULATE_SLAVE_POSITION_REQUEST			:= 196,
	CSP_CASE_STATUS_READY										:= 197,
	CSP_CASE_STATUS_RUNNING										:= 200,
	CSP_CASE_STATUS_MOVING										:= 205,
	CSP_CASE_STATUS_DISENGAGE_REQUEST							:= 210,
	CSP_CASE_STATUS_DISENGAGING									:= 211,	
	CSP_CASE_STATUS_STOP_REQUEST 								:= 500,
	CSP_CASE_STATUS_DISABLE_REQUEST 							:= 530,
	CSP_CASE_STATUS_DISABLING 									:= 540
) := CSP_CASE_STATUS_NOT_INITIALIZED;
END_TYPE

// ---- Application/CSP/Case/Discharge/csp_case_discharge_constant_struct.TcDUT
TYPE csp_case_discharge_constant_struct :
STRUCT
	(*BELT Info*)
	MIN_VELOCITY_MMpSEC:						LREAL := 100;
	MAX_VELOCITY_MMpSEC:						LREAL := 1000;
	MAX_ACCELERATION_MMpSEC2:					LREAL := 10000;
	MAX_DECELERATION_MMpSEC2:					LREAL := 10000;
	MAX_JERK_MMpSEC3:							LREAL := 1000000;
	RUNNING_ACCELERATION_MMMpSEC2:				LREAL := 3000;
	RUNNING_DECELERATION_MMpSEC2:				LREAL := 3000;
	MAX_FOLLOWING_ERROR_MM:						LREAL := 100;
	
	RUNNING_JERK_MMpSEC3:						LREAL := 1000000;
	MOTOR_MAX_VELOCITY_DEGPS:					LREAL := 9600;
	MOTOR_MAX_ACCELERATION_DEGPS2:				LREAL := 4800;
	MOTOR_MAX_DECELERATION_DEGPS2:				LREAL := 4800;
	MOTOR_MAX_JERK_DEGPS3:						LREAL := 100000000; 
	MOTOR_MAX_FOLLOWING_ERROR_DEG:				LREAL := 2;
END_STRUCT
END_TYPE

// ---- Application/CSP/Case/Discharge/csp_case_discharge_status_enum.TcDUT
TYPE csp_case_discharge_status_enum :
(
	CSP_CASE_DISCHARGE_STATUS_NOT_INITIALIZED 							:=  0,
	CSP_CASE_DISCHARGE_STATUS_DISABLED 									:=  10,
	CSP_CASE_DISCHARGE_STATUS_ENABLE_REQUEST 							:=  20,
	CSP_CASE_DISCHARGE_STATUS_ENABLING 									:=  30,
	CSP_CASE_DISCHARGE_STATUS_ENABLED 									:=  40,
	CSP_CASE_DISCHARGE_STATUS_CHANGE_OVER_MODE							:=  45,
	CSP_CASE_DISCHARGE_STATUS_HOME_REQUEST								:=  50,
	CSP_CASE_DISCHARGE_STATUS_HOMING									:=  60,
	CSP_CASE_DISCHARGE_STATUS_HOME_DONE									:=  70,
	CSP_CASE_DISCHARGE_STATUS_CALCULATING_SLAVE_POSITION				:=  90,
	CSP_CASE_DISCHARGE_STATUS_WAITING_SLAVE_ENGAGE						:= 100,
	CSP_CASE_DISCHARGE_STATUS_PHASE_REQUEST								:= 140,
	CSP_CASE_DISCHARGE_STATUS_PHASING									:= 150,
	CSP_CASE_DISCHARGE_STATUS_PHASED									:= 160,
	CSP_CASE_DISCHARGE_STATUS_CAM_ENGAGED_REQ							:= 170,
	CSP_CASE_DISCHARGE_STATUS_AXIS_ENGAGE_VERIFY						:= 180,
	CSP_CASE_DISCHARGE_STATUS_CAM_ENGAGED								:= 190,
	CSP_CASE_DISCHARGE_STATUS_CAM_TABLE_READ							:= 195,
	CSP_CASE_DISCHARGE_STATUS_CALCULATE_SLAVE_POSITION_REQUEST			:= 196,
	CSP_CASE_DISCHARGE_STATUS_READY										:= 197,
	CSP_CASE_DISCHARGE_STATUS_RUNNING									:= 200,
	CSP_CASE_DISCHARGE_STATUS_MOVING									:= 205,
	CSP_CASE_DISCHARGE_STATUS_DISENGAGE_REQUEST						:= 210,
	CSP_CASE_DISCHARGE_STATUS_DISENGAGING								:= 211,	
	CSP_CASE_DISCHARGE_STATUS_STOP_REQUEST 								:= 500,
	CSP_CASE_DISCHARGE_STATUS_DISABLE_REQUEST 							:= 530,
	CSP_CASE_DISCHARGE_STATUS_DISABLING 								:= 540
) := CSP_CASE_DISCHARGE_STATUS_NOT_INITIALIZED;
END_TYPE

// ---- Application/CSP/Case/Feed/csp_case_feed_connection_status_enum.TcDUT
TYPE csp_case_feed_connection_status_enum :
(		
	CSP_CASE_FEED_STATUS_CONNECTION_START							:= 0,
	CSP_CASE_FEED_STATUS_CONNECTION_ENGAGE							:= 10,
	CSP_CASE_FEED_STATUS_CONNECTION_ENGAGED							:= 20,
	CSP_CASE_FEED_STATUS_CONNECTION_CHECK_CHANGE_CAM				:= 30,
	CSP_CASE_FEED_STATUS_CONNECTION_CHANGE_CAM						:= 40,
	CSP_CASE_FEED_STATUS_CONNECTION_WAIT_NEW_CAM					:= 50,
	CSP_CASE_FEED_STATUS_CONNECTION_STOPPING						:= 100,
	CSP_CASE_FEED_STATUS_CONNECTION_STOPPED							:= 110,
	CSP_CASE_FEED_STATUS_CONNECTION_REJECT_STEP1					:= 201,
	CSP_CASE_FEED_STATUS_CONNECTION_REJECT_STEP2					:= 202,
	CSP_CASE_FEED_STATUS_CONNECTION_REJECT_STEP3					:= 203,
	CSP_CASE_FEED_STATUS_CONNECTION_REJECT_STEP4					:= 204,
	CSP_CASE_FEED_STATUS_CONNECTION_REJECT_STEP5					:= 205,
	CSP_CASE_FEED_STATUS_CONNECTION_REJECT_STEP6					:= 206,
	CSP_CASE_FEED_STATUS_CONNECTION_REJECT_STEP7					:= 207,
	CSP_CASE_FEED_STATUS_CONNECTION_REJECT_STEP8					:= 208,
	CSP_CASE_FEED_STATUS_CONNECTION_REJECT_STEP9					:= 209,	
	CSP_CASE_FEED_STATUS_CONNECTION_DONE 							:= 900,
	CSP_CASE_FEED_STATUS_CONNECTION_ERROR 							:= 999
) := CSP_CASE_FEED_STATUS_CONNECTION_START;
END_TYPE

// ---- Application/CSP/Case/Feed/csp_case_feed_constant_struct.TcDUT
TYPE csp_case_feed_constant_struct :
STRUCT
	(*BELT Info*)
	MIN_VELOCITY_MMpSEC:						LREAL := 100;
	MAX_VELOCITY_MMpSEC:						LREAL := 1000;
	MAX_ACCELERATION_MMpSEC2:					LREAL := 10000;
	MAX_DECELERATION_MMpSEC2:					LREAL := 10000;
	MAX_JERK_MMpSEC3:							LREAL := 1000000;
	RUNNING_ACCELERATION_MMMpSEC2:				LREAL := 3000;
	RUNNING_DECELERATION_MMpSEC2:				LREAL := 3000;
	MAX_FOLLOWING_ERROR_MM:						LREAL := 100;
	
	RUNNING_JERK_MMpSEC3:						LREAL := 1000000;
	MOTOR_MAX_VELOCITY_DEGPS:					LREAL := 9600;
	MOTOR_MAX_ACCELERATION_DEGPS2:				LREAL := 4800;
	MOTOR_MAX_DECELERATION_DEGPS2:				LREAL := 4800;
	MOTOR_MAX_JERK_DEGPS3:						LREAL := 100000000; 
	MOTOR_MAX_FOLLOWING_ERROR_DEG:				LREAL := 2;
END_STRUCT
END_TYPE

// ---- Application/CSP/Case/Feed/csp_case_feed_kinematic_constant_struct.TcDUT
TYPE csp_case_feed_kinematic_constant_struct :
STRUCT
	(*BELT Info*)
	MIN_VELOCITY_MMpSEC:						LREAL := 100;
	MAX_VELOCITY_MMpSEC:						LREAL := 1000;
	MAX_ACCELERATION_MMpSEC2:					LREAL := 10000;
	MAX_DECELERATION_MMpSEC2:					LREAL := 10000;
	MAX_JERK_MMpSEC3:							LREAL := 1000000;
	RUNNING_ACCELERATION_MMMpSEC2:				LREAL := 3000;
	RUNNING_DECELERATION_MMpSEC2:				LREAL := 3000;
	MAX_FOLLOWING_ERROR_MM:						LREAL := 100;
	
	RUNNING_JERK_MMpSEC3:						LREAL := 1000000;
	MOTOR_MAX_VELOCITY_DEGPS:					LREAL := 9600;
	MOTOR_MAX_ACCELERATION_DEGPS2:				LREAL := 4800;
	MOTOR_MAX_DECELERATION_DEGPS2:				LREAL := 4800;
	MOTOR_MAX_JERK_DEGPS3:						LREAL := 100000000; 
	MOTOR_MAX_FOLLOWING_ERROR_DEG:				LREAL := 2;
END_STRUCT
END_TYPE

// ---- Application/CSP/Case/Feed/csp_case_feed_kinematic_status_enum.TcDUT
TYPE csp_case_feed_kinematic_status_enum :
(
	CSP_CASE_FEED_KINEMATIC_STATUS_NOT_INITIALIZED 							:= 0,
	CSP_CASE_FEED_KINEMATIC_STATUS_DISABLED 								:= 10,
	CSP_CASE_FEED_KINEMATIC_STATUS_ENABLE_REQUEST 							:= 20,
	CSP_CASE_FEED_KINEMATIC_STATUS_ENABLING 								:= 30,
	CSP_CASE_FEED_KINEMATIC_STATUS_ENABLED 									:= 40,
	CSP_CASE_FEED_KINEMATIC_STATUS_CHANGE_OVER_MODE                         := 50,
    CSP_CASE_FEED_KINEMATIC_STATUS_CHANGE_OVER_MODE_DONE                    := 60,   	
	CSP_CASE_FEED_KINEMATIC_STATUS_KIN_CONFIG								:= 100,
	CSP_CASE_FEED_KINEMATIC_STATUS_JOG_ACS1									:= 101,
	CSP_CASE_FEED_KINEMATIC_STATUS_JOG_ACS2									:= 102,
	CSP_CASE_FEED_KINEMATIC_STATUS_JOG_ACS3									:= 103,
	CSP_CASE_FEED_KINEMATIC_STATUS_JOG_MCS1									:= 105,
	CSP_CASE_FEED_KINEMATIC_STATUS_JOG_MCS2									:= 106,
	CSP_CASE_FEED_KINEMATIC_STATUS_JOG_MCS3									:= 107,
	CSP_CASE_FEED_KINEMATIC_STATUS_MOVE_ACS1								:= 111,
	CSP_CASE_FEED_KINEMATIC_STATUS_MOVE_ACS2								:= 112,
	CSP_CASE_FEED_KINEMATIC_STATUS_MOVE_ACS3								:= 113,
	CSP_CASE_FEED_KINEMATIC_STATUS_MOVE_MCS1								:= 115,
	CSP_CASE_FEED_KINEMATIC_STATUS_MOVE_MCS2								:= 116,
	CSP_CASE_FEED_KINEMATIC_STATUS_MOVE_MCS3								:= 117,
	CSP_CASE_FEED_KINEMATIC_STATUS_STOP_ACS1								:= 121,
	CSP_CASE_FEED_KINEMATIC_STATUS_STOP_ACS2								:= 122,
	CSP_CASE_FEED_KINEMATIC_STATUS_STOP_ACS3								:= 123,
	CSP_CASE_FEED_KINEMATIC_STATUS_STOP_MCS1								:= 125,
	CSP_CASE_FEED_KINEMATIC_STATUS_STOP_MCS2								:= 126,
	CSP_CASE_FEED_KINEMATIC_STATUS_STOP_MCS3								:= 127,		
	CSP_CASE_FEED_KINEMATIC_STATUS_PHASE_REQUEST							:= 150,
	CSP_CASE_FEED_KINEMATIC_STATUS_PHASING									:= 160,
	CSP_CASE_FEED_KINEMATIC_STATUS_PHASED									:= 170,
	CSP_CASE_FEED_KINEMATIC_STATUS_READY_TO_ENGAGE							:= 180,
	CSP_CASE_FEED_KINEMATIC_STATUS_CAM_ENGAGED_REQ							:= 200,	
	CSP_CASE_FEED_KINEMATIC_STATUS_CAM_ENGAGED								:= 210,
	CSP_CASE_FEED_KINEMATIC_STATUS_STOP_REQUEST 							:= 500,
	CSP_CASE_FEED_KINEMATIC_STATUS_DISABLE_REQUEST 							:= 510,
	CSP_CASE_FEED_KINEMATIC_STATUS_DISABLING_KINEMATIC						:= 511,
	CSP_CASE_FEED_KINEMATIC_STATUS_DISABLING_AXIS							:= 512,
	CSP_CASE_FEED_KINEMATIC_STATUS_DISABLING 								:= 520		
) := CSP_CASE_FEED_KINEMATIC_STATUS_NOT_INITIALIZED;
END_TYPE

// ---- Application/CSP/Case/Feed/csp_case_feed_phase_status_enum.TcDUT
TYPE csp_case_feed_phase_status_enum :
(		
	CSP_CASE_FEED_STATUS_PHASE_START						:= 0,
	CSP_CASE_FEED_STATUS_PHASE_DISABLE 						:= 10,
	CSP_CASE_FEED_STATUS_PHASE_ENABLE 						:= 20,	
	CSP_CASE_FEED_STATUS_PHASE_ACTIVATE_KINEMATIC			:= 30,
	CSP_CASE_FEED_STATUS_PHASE_CALCULATE_SLAVE_POSITION		:= 40,
	CSP_CASE_FEED_STATUS_PHASE_READ_SLAVE_POSITION			:= 50,	
	CSP_CASE_FEED_STATUS_PHASE_CHECK_Y_POS					:= 51,
	CSP_CASE_FEED_STATUS_PHASE_WAIT_FOR_FOLL_SPREAD			:= 52,
	CSP_CASE_FEED_STATUS_PHASE_MOVE_SLAVE_POSITION			:= 60,
	CSP_CASE_FEED_STATUS_PHASE_MOVED_SLAVE_POSITION			:= 70,
	CSP_CASE_FEED_STATUS_PHASE_DONE 						:= 900,
	CSP_CASE_FEED_STATUS_PHASE_ERROR 						:= 999
) := CSP_CASE_FEED_STATUS_PHASE_START;
END_TYPE

// ---- Application/CSP/Case/Feed/csp_case_feed_status_enum.TcDUT
TYPE csp_case_feed_status_enum :
(
	CSP_CASE_FEED_STATUS_NOT_INITIALIZED 							:=  0,
	CSP_CASE_FEED_STATUS_DISABLED 									:=  10,
	CSP_CASE_FEED_STATUS_ENABLE_REQUEST 							:=  20,
	CSP_CASE_FEED_STATUS_ENABLING 									:=  30,
	CSP_CASE_FEED_STATUS_ENABLED 									:=  40,
	CSP_CASE_FEED_STATUS_CHANGE_OVER_MODE                           :=  60,
    CSP_CASE_FEED_STATUS_CHANGE_OVER_MODE_DONE                      :=  70,   
	CSP_CASE_FEED_STATUS_CALCULATING_SLAVE_POSITION					:=  90,
	CSP_CASE_FEED_STATUS_PHASE_REQUEST								:= 140,
	CSP_CASE_FEED_STATUS_PHASING									:= 150,
	CSP_CASE_FEED_STATUS_SLAVE_PHASING								:= 155,
	CSP_CASE_FEED_STATUS_CHECK_CARTON								:= 156,
	CSP_CASE_FEED_STATUS_CHECK_OK									:= 157,
	CSP_CASE_FEED_STATUS_PHASED										:= 160,
	CSP_CASE_FEED_STATUS_CAM_ENGAGED_REQ							:= 170,
	CSP_CASE_FEED_STATUS_AXIS_ENGAGE_VERIFY							:= 180,
	CSP_CASE_FEED_STATUS_CAM_ENGAGED								:= 190,
	CSP_CASE_FEED_STATUS_CAM_TABLE_READ								:= 195,
	CSP_CASE_FEED_STATUS_CALCULATE_SLAVE_POSITION_REQUEST			:= 196,
	CSP_CASE_FEED_STATUS_READY										:= 197,
	CSP_CASE_FEED_STATUS_RUNNING									:= 200,
	CSP_CASE_FEED_STATUS_MOVING										:= 205,
	CSP_CASE_FEED_STATUS_DISENGAGE_REQUEST							:= 210,
	CSP_CASE_FEED_STATUS_DISENGAGING								:= 211,			
	CSP_CASE_FEED_STATUS_DISENGAGED									:= 212,	
	CSP_CASE_FEED_STATUS_DISENGAGED_AND_STOPPED						:= 213,
	CSP_CASE_FEED_STATUS_REJECT_WAIT_FOLLOWER						:= 220,
	CSP_CASE_FEED_STATUS_REJECT_MOVE_BACK							:= 221,
	CSP_CASE_FEED_STATUS_REJECT_MOVED_BACK							:= 222,
	CSP_CASE_FEED_STATUS_REJECT_START_REJECT_SEQUENCE				:= 223,
	CSP_CASE_FEED_STATUS_REJECT_END_REJECT_SEQUENCE					:= 224,
	CSP_CASE_FEED_STATUS_REJECT_WAIT_NEW_CARTON						:= 225,
	CSP_CASE_FEED_STATUS_STOP_REQUEST 								:= 500,
	CSP_CASE_FEED_STATUS_DISABLE_REQUEST 							:= 530,
	CSP_CASE_FEED_STATUS_DISABLING 									:= 540
) := CSP_CASE_FEED_STATUS_NOT_INITIALIZED;
END_TYPE

// ---- Application/CSP/Case/Feed/Magazine/csp_case_feed_magazine_constant_struct.TcDUT
TYPE csp_case_feed_magazine_constant_struct :
STRUCT
	(*BELT Info*)
	MIN_VELOCITY_MMpSEC:						LREAL := 100;
	MAX_VELOCITY_MMpSEC:						LREAL := 1000;
	MAX_ACCELERATION_MMpSEC2:					LREAL := 10000;
	MAX_DECELERATION_MMpSEC2:					LREAL := 10000;
	MAX_JERK_MMpSEC3:							LREAL := 1000000;
	RUNNING_ACCELERATION_MMMpSEC2:				LREAL := 3000;
	RUNNING_DECELERATION_MMpSEC2:				LREAL := 3000;
	MAX_FOLLOWING_ERROR_MM:						LREAL := 100;
	
	RUNNING_JERK_MMpSEC3:						LREAL := 1000000;
	MOTOR_MAX_VELOCITY_DEGPS:					LREAL := 9600;
	MOTOR_MAX_ACCELERATION_DEGPS2:				LREAL := 4800;
	MOTOR_MAX_DECELERATION_DEGPS2:				LREAL := 4800;
	MOTOR_MAX_JERK_DEGPS3:						LREAL := 100000000; 
	MOTOR_MAX_FOLLOWING_ERROR_DEG:				LREAL := 2;
END_STRUCT
END_TYPE

// ---- Application/CSP/Case/Flap Control/csp_case_flap_control_connection_status_enum.TcDUT
TYPE csp_case_flap_control_connection_status_enum :
(		
	CSP_CASE_FLAP_CONTROL_STATUS_CONNECTION_START					:= 0,
	CSP_CASE_FLAP_CONTROL_STATUS_CONNECTION_ENGAGE					:= 10,
	CSP_CASE_FLAP_CONTROL_STATUS_CONNECTION_ENGAGED					:= 20,
	CSP_CASE_FLAP_CONTROL_STATUS_CONNECTION_CHECK_CHANGE_CAM			:= 30,
	CSP_CASE_FLAP_CONTROL_STATUS_CONNECTION_CHANGE_CAM				:= 40,
	CSP_CASE_FLAP_CONTROL_STATUS_CONNECTION_WAIT_NEW_CAM				:= 50,
	CSP_CASE_FLAP_CONTROL_STATUS_CONNECTION_DONE 					:= 900,
	CSP_CASE_FLAP_CONTROL_STATUS_CONNECTION_ERROR 					:= 999
) := CSP_CASE_FLAP_CONTROL_STATUS_CONNECTION_START;
END_TYPE

// ---- Application/CSP/Case/Flap Control/csp_case_flap_control_phase_status_enum.TcDUT
TYPE csp_case_flap_control_phase_status_enum :
(		
	CSP_CASE_FLAP_CONTROL_STATUS_PHASE_START							:= 0,
	CSP_CASE_FLAP_CONTROL_STATUS_PHASE_DISABLE 							:= 10,
	CSP_CASE_FLAP_CONTROL_STATUS_PHASE_ENABLE 							:= 20,	
	CSP_CASE_FLAP_CONTROL_STATUS_PHASE_ENABLED 							:= 30,
	CSP_CASE_FLAP_CONTROL_STATUS_PHASE_CALCULATE_SLAVE_POSITION_REQUEST	:= 31,
	CSP_CASE_FLAP_CONTROL_STATUS_PHASE_CALCULATING_SLAVE_POSITION		:= 32,
	CSP_CASE_FLAP_CONTROL_STATUS_PHASE_REQUESTED						:= 33,
	CSP_CASE_FLAP_CONTROL_STATUS_PHASE_PHASING							:= 34,
	CSP_CASE_FLAP_CONTROL_STATUS_PHASE_PHASED							:= 35,
	CSP_CASE_FLAP_CONTROL_STATUS_PHASE_REDEFINE							:= 40,
	CSP_CASE_FLAP_CONTROL_STATUS_PHASE_REDEFINED						:= 50,
	CSP_CASE_FLAP_CONTROL_STATUS_PHASE_DONE 							:= 900,
	CSP_CASE_FLAP_CONTROL_STATUS_PHASE_ERROR 							:= 999
) := CSP_CASE_FLAP_CONTROL_STATUS_PHASE_START;
END_TYPE

// ---- Application/CSP/Case/Flap Control/csp_case_flap_control_status_enum.TcDUT
TYPE csp_case_flap_control_status_enum :
(
	CSP_CASE_FLAP_CONTROL_STATUS_NOT_INITIALIZED 							:=  0,
	CSP_CASE_FLAP_CONTROL_STATUS_DISABLED 									:=  10,
	CSP_CASE_FLAP_CONTROL_STATUS_ENABLE_REQUEST 							:=  20,
	CSP_CASE_FLAP_CONTROL_STATUS_ENABLING 									:=  30,
	CSP_CASE_FLAP_CONTROL_STATUS_ENABLED 									:=  40,
	CSP_CASE_FLAP_CONTROL_STATUS_CHANGE_OVER_MODE							:=  45,
	CSP_CASE_FLAP_CONTROL_STATUS_CHANGE_OVER_MODE_DONE						:= 	47,
	CSP_CASE_FLAP_CONTROL_STATUS_HOME_REQUEST								:=  50,
	CSP_CASE_FLAP_CONTROL_STATUS_HOMING										:=  60,
	CSP_CASE_FLAP_CONTROL_STATUS_HOME_DONE									:=  70,
	CSP_CASE_FLAP_CONTROL_STATUS_CALCULATING_SLAVE_POSITION					:=  90,
	CSP_CASE_FLAP_CONTROL_STATUS_WAITING_SLAVE_ENGAGE						:= 100,
	CSP_CASE_FLAP_CONTROL_STATUS_WAITING_SLAVE_ENGAGE_2						:= 120,
	CSP_CASE_FLAP_CONTROL_STATUS_PHASE_REQUEST								:= 140,
	CSP_CASE_FLAP_CONTROL_STATUS_PHASING									:= 150,
	CSP_CASE_FLAP_CONTROL_STATUS_PHASED										:= 160,
	CSP_CASE_FLAP_CONTROL_STATUS_CAM_ENGAGED_REQ							:= 170,
	CSP_CASE_FLAP_CONTROL_STATUS_AXIS_ENGAGE_VERIFY							:= 180,
	CSP_CASE_FLAP_CONTROL_STATUS_CAM_ENGAGED								:= 190,
	CSP_CASE_FLAP_CONTROL_STATUS_CAM_TABLE_READ								:= 195,
	CSP_CASE_FLAP_CONTROL_STATUS_CALCULATE_SLAVE_POSITION_REQUEST			:= 196,
	CSP_CASE_FLAP_CONTROL_STATUS_READY										:= 197,
	CSP_CASE_FLAP_CONTROL_STATUS_RUNNING									:= 200,
	CSP_CASE_FLAP_CONTROL_STATUS_MOVING										:= 205,
	CSP_CASE_FLAP_CONTROL_STATUS_DISENGAGE_REQUEST							:= 210,
	CSP_CASE_FLAP_CONTROL_STATUS_DISENGAGING								:= 211,	
	
	
	CSP_CASE_FLAP_CONTROL_STATUS_STOP_REQUEST 								:= 500,
	CSP_CASE_FLAP_CONTROL_STATUS_DISABLE_REQUEST 							:= 530,
	CSP_CASE_FLAP_CONTROL_STATUS_DISABLING 									:= 540
) := CSP_CASE_FLAP_CONTROL_STATUS_NOT_INITIALIZED;
END_TYPE

// ---- Application/CSP/Case/Glue/csp_case_glue_status_enum.TcDUT
TYPE csp_case_glue_status_enum :
(
	CSP_CASE_GLUE_STATUS_INIT 							:=  0,
	CSP_CASE_GLUE_STATUS_PURGE_ACTIVATE					:=  100,
	CSP_CASE_GLUE_STATUS_PURGE_RUNNING 					:=  200,
	CSP_CASE_GLUE_STATUS_PURGE_WAITING_DEACTIVATE		:=  300,
	CSP_CASE_GLUE_STATUS_RUNNING						:=  400
) := CSP_CASE_GLUE_STATUS_INIT;
END_TYPE

// ---- Application/CSP/Case/Loader/csp_case_loader_constant_struct.TcDUT
TYPE csp_case_loader_constant_struct :
STRUCT
	(*BELT Info*)
	MIN_VELOCITY_MMpSEC:						LREAL := 100;
	MAX_VELOCITY_MMpSEC:						LREAL := 1000;
	MAX_ACCELERATION_MMpSEC2:					LREAL := 10000;
	MAX_DECELERATION_MMpSEC2:					LREAL := 10000;
	MAX_JERK_MMpSEC3:							LREAL := 1000000;
	RUNNING_ACCELERATION_MMMpSEC2:				LREAL := 3000;
	RUNNING_DECELERATION_MMpSEC2:				LREAL := 3000;
	MAX_FOLLOWING_ERROR_MM:						LREAL := 100;
	
	RUNNING_JERK_MMpSEC3:						LREAL := 1000000;
	MOTOR_MAX_VELOCITY_DEGPS:					LREAL := 9600;
	MOTOR_MAX_ACCELERATION_DEGPS2:				LREAL := 4800;
	MOTOR_MAX_DECELERATION_DEGPS2:				LREAL := 4800;
	MOTOR_MAX_JERK_DEGPS3:						LREAL := 100000000; 
	MOTOR_MAX_FOLLOWING_ERROR_DEG:				LREAL := 2;
END_STRUCT
END_TYPE

// ---- Application/CSP/Case/Loader/csp_case_loader_rfid_status_enum.TcDUT
TYPE csp_case_loader_rfid_status_enum :
(
	CSP_CASE_LOADER_RFID_STATUS_START 							:= 1,
	CSP_CASE_LOADER_RFID_STATUS_CHECK_AXIS_POS					:= 5,
	CSP_CASE_LOADER_RFID_STATUS_DISABLE_AXIS					:= 10,
	CSP_CASE_LOADER_RFID_STATUS_ENABLE_AXIS						:= 20,
	CSP_CASE_LOADER_RFID_STATUS_ENABLE_CROSSPUSHERS				:= 21,
	CSP_CASE_LOADER_RFID_STATUS_MOVE_CROSSPUSHERS				:= 22,
	CSP_CASE_LOADER_RFID_VERIFY_CROSSPUSHERS_CLEAR				:= 25,
	CSP_CASE_LOADER_RFID_STATUS_MOVE_AXIS_TO_POS				:= 30,
	CSP_CASE_LOADER_RFID_STATUS_VERIFY_AXIS_POS					:= 40,
	
	CSP_CASE_LOADER_RFID_STATUS_CHECK_READ_WRITE				:= 50,
	
	CSP_CASE_LOADER_RFID_STATUS_READ_START						:= 100,
	CSP_CASE_LOADER_RFID_STATUS_READ_CHECK_RESULT				:= 110,
	CSP_CASE_LOADER_RFID_STATUS_READ_DONE						:= 120,
	
	CSP_CASE_LOADER_RFID_STATUS_WRITE_START						:= 200,
	CSP_CASE_LOADER_RFID_STATUS_WAIT_WRITE						:= 210,
	CSP_CASE_LOADER_RFID_STATUS_WRITE_DONE						:= 220,
	
	
	CSP_CASE_LOADER_RFID_STATUS_WAITING							:= 900
) := CSP_CASE_LOADER_RFID_STATUS_WAITING;
END_TYPE

// ---- Application/CSP/Case/Loader/csp_case_phasing_enum.TcDUT
TYPE csp_case_phasing_enum :
(
	CSP_CASE_PHASING_START							:= 1,
	//CSP_CASE_PHASING_CHECK_ALL_INTERFERENCE			:= 10,
	CSP_CASE_PHASING_CHECK_LEADING_MINOR			:= 20,
	CSP_CASE_PHASING_CHECK_LOADER_GUIDES			:= 30,
	CSP_CASE_PHASING_CHECK_LOADER					:= 40,
	CSP_CASE_PHASING_CHECK_FOLLOWER					:= 50,
	
	CSP_CASE_PHASING_MOVE_GUIDES					:= 100,
	CSP_CASE_PHASING_REORDER_GUIDES					:= 105,
	CSP_CASE_PHASING_MOVE_DOWNSTREAM_GUIDE			:= 110,
	CSP_CASE_PHASING_MOVE_DOWNSTREAM_GUIDE_OUT		:= 115,
	CSP_CASE_PHASING_MOVE_UPSTREAM_GUIDE			:= 120,
	CSP_CASE_PHASING_MOVE_UPSTREAM_GUIDE_OUT		:= 125,
	CSP_CASE_PHASING_GUIDES_OUT						:= 127,
	CSP_CASE_PHASING_GUIDE_MOVE_COMPLETE			:= 130,
	
	CSP_CASE_PHASING_MOVE_LOADER					:= 200,
	CSP_CASE_PHASING_MOVE_LOADER_COMPLETE			:= 210,
	
	CSP_CASE_PHASING_MOVE_FOLLOWER					:= 300,
	CSP_CASE_PHASING_MOVE_FOLLOWER_COMPLETE			:= 310,
	
	CSP_CASE_PHASING_DONE							:= 900,
	CSP_CASE_PHASING_ERROR							:= 999
) := CSP_CASE_PHASING_DONE;
END_TYPE

// ---- Application/CSP/Case/Loader/csp_case_loader_status_enum.TcDUT
TYPE csp_case_loader_status_enum :
(
	CSP_CASE_LOADER_STATUS_NOT_INITIALIZED 							:=  0,
	CSP_CASE_LOADER_STATUS_DISABLED 								:=  10,
	CSP_CASE_LOADER_STATUS_ENABLE_REQUEST 							:=  20,
	CSP_CASE_LOADER_STATUS_ENABLING 								:=  30,
	CSP_CASE_LOADER_STATUS_ENABLED 									:=  40,
	CSP_CASE_LOADER_STATUS_CHANGE_OVER_MODE							:=  45,
	CSP_CASE_LOADER_STATUS_ENABLE_CROSSPUSHERS						:=  46,
	CSP_CASE_LOADER_STATUS_MOVE_CROSSPUSHERS						:=  47,
	CSP_CASE_LOADER_STATUS_VERIFY_CROSSPUSHERS_CLEAR				:=  48,
	CSP_CASE_LOADER_STATUS_MOVE_AXIS_TO_POS							:=  49,
	CSP_CASE_LOADER_STATUS_HOME_REQUEST								:=  50,
	CSP_CASE_LOADER_STATUS_HOMING									:=  60,
	CSP_CASE_LOADER_STATUS_HOME_DONE								:=  70,
	CSP_CASE_LOADER_STATUS_LENGTH_MOVE_TO_CLEAR_POS					:=  80,
	CSP_CASE_LOADER_STATUS_LENGTH_MOVING_TO_CLEAR_POS				:=  85,
	CSP_CASE_LOADER_STATUS_LENGTH_WAITING_FOR_GUIDES_TO_PHASE		:=  87,
	CSP_CASE_LOADER_STATUS_CALCULATING_SLAVE_POSITION				:=  90,
	CSP_CASE_LOADER_STATUS_CALCULATING_MASTER_POSITION				:=  91,
	CSP_CASE_LOADER_STATUS_WAITING_SLAVE_ENGAGE						:= 100,
	CSP_CASE_LOADER_STATUS_WAITING_MASTER_ENGAGE					:= 101,
	CSP_CASE_LOADER_STATUS_LOADER_PLATE_PHASE_REQUIRED				:= 130,
	CSP_CASE_LOADER_STATUS_PHASE_REQUEST							:= 140,
	CSP_CASE_LOADER_STATUS_PHASING									:= 150,
	CSP_CASE_LOADER_STATUS_PHASED									:= 160,
	CSP_CASE_LOADER_STATUS_CAM_ENGAGED_REQ							:= 170,
	CSP_CASE_LOADER_STATUS_AXIS_ENGAGE_VERIFY						:= 180,
	CSP_CASE_LOADER_STATUS_CAM_ENGAGED								:= 190,
	CSP_CASE_LOADER_STATUS_CAM_TABLE_READ							:= 195,
	CSP_CASE_LOADER_STATUS_CALCULATE_SLAVE_POSITION_REQUEST			:= 196,
	CSP_CASE_LOADER_STATUS_READY									:= 197,
	CSP_CASE_LOADER_STATUS_RUNNING									:= 200,
	CSP_CASE_LOADER_STATUS_MOVING									:= 205,
	CSP_CASE_LOADER_STATUS_DISENGAGE_REQUEST						:= 210,
	CSP_CASE_LOADER_STATUS_DISENGAGING								:= 211,	
	CSP_CASE_LOADER_STATUS_STOP_REQUEST 							:= 500,
	CSP_CASE_LOADER_STATUS_DISABLE_REQUEST 							:= 530,
	CSP_CASE_LOADER_STATUS_DISABLING 								:= 540,
	
	CSP_CASE_LOADER_STATUS_IMMEDIATE_DWELL_FOR_CASE_ALREADY_LOADED	:= 560,
	CSP_CASE_LOADER_STATUS_WAIT_FOR_REJECT_DONE						:= 565,
	CSP_CASE_LOADER_STATUS_WAIT_FOR_STACK_AT_LOADER					:= 570,
	CSP_CASE_LOADER_STATUS_FINISH_LOAD_CYCLE						:= 575,
	CSP_CASE_LOADER_STATUS_WAIT_FOR_NEW_LOAD						:= 580,
	CSP_CASE_LOADER_STATUS_LOAD_COMPLETE							:= 585,
	
	CSP_CASE_LOADER_STATUS_IMMEDIATE_DWELL_FOR_REJECT				:= 600,
	CSP_CASE_LOADER_STATUS_WAIT_FOR_REJECT_COMPLETE					:= 610,
	CSP_CASE_LOADER_STATUS_WAIT_FOR_LOAD							:= 620,
	CSP_CASE_LOADER_STATUS_VERIFY_SLAVES_ENGAGED					:= 630,
	CSP_CASE_LOADER_STATUS_RUN_LOAD_CYCLE							:= 640,
	CSP_CASE_LOADER_STATUS_ENGAGE_TO_CASE_VM						:= 650,
	
	CSP_CASE_LOADER_STATUS_IMMEDIATE_DISENGAGE_THEN_WAIT_CAM		:= 700,
	CSP_CASE_LOADER_STATUS_IMMEDIATE_DISENGAGE_CHECK_ZERO			:= 701,
	CSP_CASE_LOADER_STATUS_IMMEDIATE_DISENGAGE_MOVE_TO_ZERO			:= 702,
	CSP_CASE_LOADER_STATUS_IMMEDIATE_DISENGAGE_WAIT_MOVE			:= 703
	
) := CSP_CASE_LOADER_STATUS_NOT_INITIALIZED;
END_TYPE

// ---- Application/CSP/Case/Main/statistics/csp_case_main_statistics_debug_struct.TcDUT
TYPE csp_case_main_statistics_debug_struct :
STRUCT
	step_id:				INT;
	reject_reason:			DWORD;
	status:					DWORD;
	//item_has:				INT;
END_STRUCT
END_TYPE

// ---- Application/CSP/Case/Top Rail/Squaring/csp_case_topRail_squaring_status_enum.TcDUT
TYPE csp_case_topRail_squaring_status_enum :
(
	CSP_CASE_TOPRAIL_SQUARING_STATUS_NOT_INITIALIZED 							:=  0,
	CSP_CASE_TOPRAIL_SQUARING_STATUS_DISABLED 									:=  10,
	CSP_CASE_TOPRAIL_SQUARING_STATUS_ENABLE_REQUEST 							:=  20,
	CSP_CASE_TOPRAIL_SQUARING_STATUS_ENABLING 									:=  30,
	CSP_CASE_TOPRAIL_SQUARING_STATUS_ENABLED 									:=  40,
	CSP_CASE_TOPRAIL_SQUARING_STATUS_CHANGE_OVER_MODE						   	:=  45,
	CSP_CASE_TOPRAIL_SQUARING_STATUS_HOME_REQUEST								:=  50,
	CSP_CASE_TOPRAIL_SQUARING_STATUS_HOMING										:=  60,
	CSP_CASE_TOPRAIL_SQUARING_STATUS_HOME_DONE									:=  70,
	CSP_CASE_TOPRAIL_SQUARING_STATUS_CALCULATING_SLAVE_POSITION					:=  90,
	CSP_CASE_TOPRAIL_SQUARING_STATUS_WAITING_SLAVE_ENGAGE						:= 100,
	CSP_CASE_TOPRAIL_SQUARING_STATUS_PHASE_REQUEST								:= 140,
	CSP_CASE_TOPRAIL_SQUARING_STATUS_PHASING									:= 150,
	CSP_CASE_TOPRAIL_SQUARING_STATUS_PHASED										:= 160,
	CSP_CASE_TOPRAIL_SQUARING_STATUS_CAM_ENGAGED_REQ							:= 170,
	CSP_CASE_TOPRAIL_SQUARING_STATUS_AXIS_ENGAGE_VERIFY							:= 180,
	CSP_CASE_TOPRAIL_SQUARING_STATUS_CAM_ENGAGED								:= 190,
	CSP_CASE_TOPRAIL_SQUARING_STATUS_CAM_TABLE_READ								:= 195,
	CSP_CASE_TOPRAIL_SQUARING_STATUS_CALCULATE_SLAVE_POSITION_REQUEST			:= 196,
	CSP_CASE_TOPRAIL_SQUARING_STATUS_READY										:= 197,
	CSP_CASE_TOPRAIL_SQUARING_STATUS_RUNNING									:= 200,
	CSP_CASE_TOPRAIL_SQUARING_STATUS_MOVING										:= 205,
	CSP_CASE_TOPRAIL_SQUARING_STATUS_DISENGAGE_REQUEST							:= 210,
	CSP_CASE_TOPRAIL_SQUARING_STATUS_DISENGAGING								:= 211,	
	CSP_CASE_TOPRAIL_SQUARING_STATUS_STOP_REQUEST 								:= 500,
	CSP_CASE_TOPRAIL_SQUARING_STATUS_DISABLE_REQUEST 							:= 530,
	CSP_CASE_TOPRAIL_SQUARING_STATUS_DISABLING 									:= 540
	) := CSP_CASE_TOPRAIL_SQUARING_STATUS_NOT_INITIALIZED;
END_TYPE

// ---- Application/CSP/Case/Top Rail/Squaring/csp_case_topRail_squaring_struct.TcDUT
TYPE csp_case_topRail_squaring_struct :
STRUCT
	(*BELT Info*)
	MIN_VELOCITY_MMpSEC:						LREAL := 100;
	MAX_VELOCITY_MMpSEC:						LREAL := 1000;
	MAX_ACCELERATION_MMpSEC2:					LREAL := 10000;
	MAX_DECELERATION_MMpSEC2:					LREAL := 10000;
	MAX_JERK_MMpSEC3:							LREAL := 1000000;
	RUNNING_ACCELERATION_MMMpSEC2:				LREAL := 3000;
	RUNNING_DECELERATION_MMpSEC2:				LREAL := 3000;
	MAX_FOLLOWING_ERROR_MM:						LREAL := 100;
	
	RUNNING_JERK_MMpSEC3:						LREAL := 1000000;
	MOTOR_MAX_VELOCITY_DEGPS:					LREAL := 9600;
	MOTOR_MAX_ACCELERATION_DEGPS2:				LREAL := 4800;
	MOTOR_MAX_DECELERATION_DEGPS2:				LREAL := 4800;
	MOTOR_MAX_JERK_DEGPS3:						LREAL := 100000000; 
	MOTOR_MAX_FOLLOWING_ERROR_DEG:				LREAL := 2;
END_STRUCT
END_TYPE

// ---- Application/CSP/Case/Transport/csp_case_transport_constant_struct.TcDUT
TYPE csp_case_transport_constant_struct :
STRUCT
	(*BELT Info*)
	MIN_VELOCITY_MMpSEC:						LREAL := 100;
	MAX_VELOCITY_MMpSEC:						LREAL := 1000;
	MAX_ACCELERATION_MMpSEC2:					LREAL := 10000;
	MAX_DECELERATION_MMpSEC2:					LREAL := 10000;
	MAX_JERK_MMpSEC3:							LREAL := 1000000;
	RUNNING_ACCELERATION_MMMpSEC2:				LREAL := 3000;
	RUNNING_DECELERATION_MMpSEC2:				LREAL := 3000;
	MAX_FOLLOWING_ERROR_MM:						LREAL := 100;
	
	RUNNING_JERK_MMpSEC3:						LREAL := 1000000;
	MOTOR_MAX_VELOCITY_DEGPS:					LREAL := 9600;
	MOTOR_MAX_ACCELERATION_DEGPS2:				LREAL := 4800;
	MOTOR_MAX_DECELERATION_DEGPS2:				LREAL := 4800;
	MOTOR_MAX_JERK_DEGPS3:						LREAL := 100000000; 
	MOTOR_MAX_FOLLOWING_ERROR_DEG:				LREAL := 2;
END_STRUCT
END_TYPE

// ---- Application/CSP/Case/Transport/csp_case_transport_status_enum.TcDUT
TYPE csp_case_transport_status_enum :
(
	CSP_CASE_TRANSPORT_STATUS_NOT_INITIALIZED 							:=  0,
	CSP_CASE_TRANSPORT_STATUS_DISABLED 									:=  10,
	CSP_CASE_TRANSPORT_STATUS_ENABLE_REQUEST 							:=  20,
	CSP_CASE_TRANSPORT_STATUS_ENABLING 									:=  30,
	CSP_CASE_TRANSPORT_STATUS_ENABLED 									:=  40,
	CSP_CASE_TRANSPORT_STATUS_CHANGE_OVER_MODE							:=  45,
	CSP_CASE_TRANSPORT_STATUS_HOME_REQUEST								:=  50,
	CSP_CASE_TRANSPORT_STATUS_HOMING									:=  60,
	CSP_CASE_TRANSPORT_STATUS_HOME_DONE									:=  70,
	CSP_CASE_TRANSPORT_STATUS_CALCULATING_SLAVE_POSITION				:=  90,
	CSP_CASE_TRANSPORT_STATUS_CALCULATING_MASTER_POSITION				:=  91,
	CSP_CASE_TRANSPORT_STATUS_WAITING_SLAVE_ENGAGE						:= 100,
	CSP_CASE_TRANSPORT_STATUS_WAITING_MASTER_ENGAGE						:= 101,
	CSP_CASE_TRANSPORT_STATUS_PHASE_REQUEST								:= 140,
	CSP_CASE_TRANSPORT_STATUS_PHASING									:= 150,
	CSP_CASE_TRANSPORT_STATUS_PHASED									:= 160,
	CSP_CASE_TRANSPORT_STATUS_CAM_ENGAGED_REQ							:= 170,
	CSP_CASE_TRANSPORT_STATUS_AXIS_ENGAGE_VERIFY						:= 180,
	CSP_CASE_TRANSPORT_STATUS_CAM_ENGAGED								:= 190,
	CSP_CASE_TRANSPORT_STATUS_CAM_TABLE_READ							:= 195,
	CSP_CASE_TRANSPORT_STATUS_CALCULATE_SLAVE_POSITION_REQUEST			:= 196,
	CSP_CASE_TRANSPORT_STATUS_READY										:= 197,
	CSP_CASE_TRANSPORT_STATUS_RUNNING									:= 200,
	CSP_CASE_TRANSPORT_STATUS_MOVING									:= 205,
	CSP_CASE_TRANSPORT_STATUS_DISENGAGE_REQUEST							:= 210,
	CSP_CASE_TRANSPORT_STATUS_DISENGAGING								:= 211,	
	CSP_CASE_TRANSPORT_STATUS_STOP_REQUEST 								:= 500,
	CSP_CASE_TRANSPORT_STATUS_DISABLE_REQUEST 							:= 530,
	CSP_CASE_TRANSPORT_STATUS_DISABLING 								:= 540,
	
	CSP_CASE_TRANSPORT_STATUS_RECOVERY_CAM_ENGAGED_REQ					:= 305,
	CSP_CASE_TRANSPORT_STATUS_DISENGAGE_REJECT							:= 300,
	CSP_CASE_TRANSPORT_STATUS_REJECT_ABS_STEP_1							:= 301,
	CSP_CASE_TRANSPORT_STATUS_REJECT_ABS_STEP_2							:= 302,
	CSP_CASE_TRANSPORT_STATUS_REJECT_ABS_STEP_3							:= 303,
	CSP_CASE_TRANSPORT_STATUS_REJECT_ABS_STEP_4							:= 304	
	
) := CSP_CASE_TRANSPORT_STATUS_NOT_INITIALIZED;
END_TYPE

// ---- Application/CSP/csp_retain_data_struct.TcDUT
(*********************************** G.D S.p.A. - Technical Department ***********************************
============= PROGRAM INFO ============


============= DESCRIPTION =============


============= REVISIONS ===============
Date		Version	 	Author      	Description             
----------	-------		------------  	--------------------------------------------
2019/04/24 	0000.00	 	CEC 			Creation of the PRG

**********************************************************************************************************)

TYPE csp_retain_data_struct :
STRUCT
	motorization_axis_position:		LREAL;
	carton_erected:					BOOL;
END_STRUCT
END_TYPE

// ---- Application/CSP/Customer Interface/csp_customerInterfaces_casePacker.TcDUT
(*********************************** G.D S.p.A. - Technical Department ***********************************
============= PROGRAM INFO ============
FOLDER:             TBD
MACHINES INVOLVED:  TBD 

============= DESCRIPTION =============
Machine declaration

============= REVISIONS ===============
Date		Version	 	Author      	Description             
----------	-------		------------  	--------------------------------------------
2019/03/27 	0000.00	 	CEC 			Creation of the PRG

**********************************************************************************************************)

TYPE csp_customerInterfaces_casePacker :
STRUCT
	
	Status:						csp_customerInterfaces_casePackerStatus;
	Start:						csp_customerInterfaces_casePackerStart;
	Production:					csp_customerInterfaces_casePackerProduction;
	CaseBlanks:					csp_customerInterfaces_casePackerCaseBlanks;	
	Labels:						csp_customerInterfaces_casePackerLabels;
	CtCall:						csp_customerInterfaces_casePackerCtCall;
	Dock:						ARRAY[1..3] OF csp_customerInterfaces_casePackerDock;
															
END_STRUCT
END_TYPE

// ---- Application/CSP/Customer Interface/csp_customerInterfaces_casePackerCaseBlanks.TcDUT
(*********************************** G.D S.p.A. - Technical Department ***********************************
============= PROGRAM INFO ============
FOLDER:             TBD
MACHINES INVOLVED:  TBD 

============= DESCRIPTION =============
Machine declaration

============= REVISIONS ===============
Date		Version	 	Author      	Description             
----------	-------		------------  	--------------------------------------------
2019/03/27 	0000.00	 	CEC 			Creation of the PRG

**********************************************************************************************************)

TYPE csp_customerInterfaces_casePackerCaseBlanks :
STRUCT
	
